        f_MessageSet(_stMsg);
      END_IF
    END_IF
END_CASE
//---------------------------------------------------------------------------------------
//  get config data
//    - NCI: X,Y,Z and helper axis Ids
//---------------------------------------------------------------------------------------
CASE _eState
OF
  E_PROGRESS.PROGRESS_BUSY:
    _AxisIdentity             := _stConfiguration.PortalConfig.AxisIdentity;
    _eState                   := E_PROGRESS.PROGRESS_PREPARE;
END_CASE
//---------------------------------------------------------------------------------------
//  check config data and initialize NCI Group
//    --> ST_AXIS_GROUP_INFO: data struct for plausibility checks on NCI Group
//---------------------------------------------------------------------------------------
CASE _eState
OF
  E_PROGRESS.PROGRESS_PREPARE:
    _eRslt                    := Unit_StartUp(TRUE);
    
    IF (_eRslt = E_PROGRESS.PROGRESS_ERROR)
    THEN
      // base class did the messaging
      // exit with error
      _eStateError            := _eState;
      _eState                 := E_PROGRESS.PROGRESS_ERROR;
      _eRslt                  := Unit_StartUp(FALSE);   // clear method

    ELSIF (_eRslt = E_PROGRESS.PROGRESS_DONE)
    THEN
      // startup of NCI successful
      // next states are intended for customization
      _eState                 := E_PROGRESS.PROGRESS_STARTUP;
      _eRslt                  := Unit_StartUp(FALSE);   // clear method
    END_IF
END_CASE
//---------------------------------------------------------------------------------------
//---------------------------------------------------------------------------------------
CASE _eState
OF
  E_PROGRESS.PROGRESS_STARTUP:
      // simply an inexpensive placeholder to customize initialization to your needs
      _eState                 := E_PROGRESS.PROGRESS_CHECK;
END_CASE
//---------------------------------------------------------------------------------------
//---------------------------------------------------------------------------------------
CASE _eState
OF
  E_PROGRESS.PROGRESS_CHECK:
      _eState                 := E_PROGRESS.PROGRESS_OCCUPIED;
END_CASE
//---------------------------------------------------------------------------------------
//---------------------------------------------------------------------------------------
CASE _eState
OF
  E_PROGRESS.PROGRESS_OCCUPIED:
      _eState                 := E_PROGRESS.PROGRESS_WORKING;
END_CASE
//---------------------------------------------------------------------------------------
//---------------------------------------------------------------------------------------
CASE _eState
OF
  E_PROGRESS.PROGRESS_WORKING:
    _eState                   := E_PROGRESS.PROGRESS_DONE;

    IF (_MessageLevel > E_MessageType.eMessageError)
    THEN
      _stMsg.eType            := E_MessageType.eMessageInfo;
      _stMsg.eSubdevice       := e_Subdevice.JobControl_Init;
      _stMsg.iErrorNumber     := _eState;
      _stMsg.sText            := concat(': ', TO_STRING(_eState));
    
      f_MessageSet(_stMsg);
    END_IF
END_CASE


Job_Init                      := _eState;
END_METHOD

METHOD Job_Reset  : E_PROGRESS
VAR_INPUT
  Execute         : BOOL;
END_VAR
VAR_INST
  _eRslt,
  _eStateError,
  _eState         : E_PROGRESS;
END_VAR
//---------------------------------------------------------------------------------------
//---------------------------------------------------------------------------------------
IF NOT Execute THEN _eState   := _eStateError     := E_PROGRESS.PROGRESS_INIT;  RETURN; END_IF
//---------------------------------------------------------------------------------------
IF NOT Check() THEN Job_Reset := _eState          := E_PROGRESS.PROGRESS_ERROR; RETURN; END_IF
//---------------------------------------------------------------------------------------
//---------------------------------------------------------------------------------------
CASE _eState 
of
  E_PROGRESS.PROGRESS_INIT:
    IF Execute
    THEN
      _eState                 := E_PROGRESS.PROGRESS_BUSY;
      _eRslt                  := Unit_Reset(FALSE);   // clear method

      IF (_MessageLevel > E_MessageType.eMessageError)
      THEN
        _stMsg.eType          := E_MessageType.eMessageInfo;
        _stMsg.eSubdevice     := e_Subdevice.JobControl_Reset;
        _stMsg.iErrorNumber   := _eState;
        _stMsg.sText          := concat(': ', TO_STRING(_eState));
      
        f_MessageSet(_stMsg);
      END_IF
    END_IF
END_CASE
//---------------------------------------------------------------------------------------
//  clear axis and NCI
//    - NCI: X,Y,Z and helper axis Ids
//---------------------------------------------------------------------------------------
CASE _eState
OF
  E_PROGRESS.PROGRESS_BUSY:
    _eRslt                    := Unit_Reset(TRUE);
    
    IF (_eRslt = E_PROGRESS.PROGRESS_ERROR)
    THEN
      // base class did the messaging
      // exit with error
      _eStateError            := _eState;
      _eState                 := E_PROGRESS.PROGRESS_ERROR;
      _eRslt                  := Unit_Reset(FALSE);   // clear method

    ELSIF (_eRslt = E_PROGRESS.PROGRESS_DONE)
    THEN
      // reset of axis and NCI successful
      // next states are intended for customization
      _eState                 := E_PROGRESS.PROGRESS_STARTUP;
      _eRslt                  := Unit_Reset(FALSE);   // clear method
    END_IF
END_CASE
//---------------------------------------------------------------------------------------
//---------------------------------------------------------------------------------------
CASE _eState
OF
  E_PROGRESS.PROGRESS_PREPARE:
      // simply an inexpensive placeholder to customize initialization to your needs
      _eState                 := E_PROGRESS.PROGRESS_STARTUP;
END_CASE
//---------------------------------------------------------------------------------------
//---------------------------------------------------------------------------------------
CASE _eState
OF
  E_PROGRESS.PROGRESS_STARTUP:
      // simply an inexpensive placeholder to customize initialization to your needs
      _eState                 := E_PROGRESS.PROGRESS_CHECK;
END_CASE
//---------------------------------------------------------------------------------------
//---------------------------------------------------------------------------------------
CASE _eState
OF
  E_PROGRESS.PROGRESS_CHECK:
      _eState                 := E_PROGRESS.PROGRESS_OCCUPIED;
END_CASE
//---------------------------------------------------------------------------------------
//---------------------------------------------------------------------------------------
CASE _eState
OF
  E_PROGRESS.PROGRESS_OCCUPIED:
      _eState                 := E_PROGRESS.PROGRESS_WORKING;
END_CASE
//---------------------------------------------------------------------------------------
//---------------------------------------------------------------------------------------
CASE _eState
OF
  E_PROGRESS.PROGRESS_WORKING:
    _eState                   := E_PROGRESS.PROGRESS_DONE;

    IF (_MessageLevel > E_MessageType.eMessageError)
    THEN
      _stMsg.eType            := E_MessageType.eMessageInfo;
      _stMsg.eSubdevice       := e_Subdevice.JobControl_Reset;
      _stMsg.iErrorNumber     := _eState;
      _stMsg.sText            := concat(': ', TO_STRING(_eState));
    
      f_MessageSet(_stMsg);
    END_IF
END_CASE


Job_Reset                     := _eState;
END_METHOD

METHOD Job_Rinse  : E_PROGRESS
VAR_INPUT
  Execute         : BOOL;
END_VAR
VAR_INST
  _eRslt,
  _eStateError,
  _eState         : E_PROGRESS;
END_VAR
//---------------------------------------------------------------------------------------
//---------------------------------------------------------------------------------------
IF NOT Execute THEN _eState   := _eStateError     := E_PROGRESS.PROGRESS_INIT;  RETURN; END_IF
//---------------------------------------------------------------------------------------
IF NOT Check() THEN Job_Rinse := _eState          := E_PROGRESS.PROGRESS_ERROR; RETURN; END_IF
//---------------------------------------------------------------------------------------
//---------------------------------------------------------------------------------------
CASE _eState 
of
  E_PROGRESS.PROGRESS_INIT:
    IF Execute
    THEN
      _eState                 := E_PROGRESS.PROGRESS_BUSY;
      // get job data at start
      _JobData                := _stConfiguration.JobConfig.ParameterRinse;
      _eRslt                  := Unit_Job(FALSE, _JobData);   // clear method

      IF (_MessageLevel > E_MessageType.eMessageError)
      THEN
        _stMsg.eType          := E_MessageType.eMessageInfo;
        _stMsg.eSubdevice     := e_Subdevice.JobControl_Rinse;
        _stMsg.iErrorNumber   := _eState;
        _stMsg.sText          := concat(': ', TO_STRING(_eState));
      
        f_MessageSet(_stMsg);
      END_IF
    END_IF
END_CASE
//---------------------------------------------------------------------------------------
//  move PtP axis
//    - X,Y,Z
//---------------------------------------------------------------------------------------
CASE _eState
OF
  E_PROGRESS.PROGRESS_BUSY:
    _eRslt                    := Unit_Job(TRUE, _JobData);
    
    IF (_eRslt = E_PROGRESS.PROGRESS_ERROR)
    THEN
      // base class did the messaging
      // exit with error
      _eStateError            := _eState;
      _eState                 := E_PROGRESS.PROGRESS_ERROR;
      _eRslt                  := Unit_Job(FALSE, _JobData);   // clear method

    ELSIF (_eRslt = E_PROGRESS.PROGRESS_DONE)
    THEN
      // move of axis to home positions successful
      // next states are intended for customization
      _eState                 := E_PROGRESS.PROGRESS_STARTUP;
      _eRslt                  := Unit_Job(FALSE, _JobData);   // clear method
    END_IF
END_CASE
//---------------------------------------------------------------------------------------
//---------------------------------------------------------------------------------------
CASE _eState
OF
  E_PROGRESS.PROGRESS_PREPARE:
      // simply an inexpensive placeholder to customize initialization to your needs
      _eState                 := E_PROGRESS.PROGRESS_STARTUP;
END_CASE
//---------------------------------------------------------------------------------------
//---------------------------------------------------------------------------------------
CASE _eState
OF
  E_PROGRESS.PROGRESS_STARTUP:
      // simply an inexpensive placeholder to customize initialization to your needs
      _eState                 := E_PROGRESS.PROGRESS_CHECK;
END_CASE
//---------------------------------------------------------------------------------------
//---------------------------------------------------------------------------------------
CASE _eState
OF
  E_PROGRESS.PROGRESS_CHECK:
      _eState                 := E_PROGRESS.PROGRESS_OCCUPIED;
END_CASE
//---------------------------------------------------------------------------------------
//---------------------------------------------------------------------------------------
CASE _eState
OF
  E_PROGRESS.PROGRESS_OCCUPIED:
      _eState                 := E_PROGRESS.PROGRESS_WORKING;
END_CASE
//---------------------------------------------------------------------------------------
//---------------------------------------------------------------------------------------
CASE _eState
OF
  E_PROGRESS.PROGRESS_WORKING:
    _eState                   := E_PROGRESS.PROGRESS_DONE;

    IF (_MessageLevel > E_MessageType.eMessageError)
    THEN
      _stMsg.eType            := E_MessageType.eMessageInfo;
      _stMsg.eSubdevice       := e_Subdevice.JobControl_Rinse;
      _stMsg.iErrorNumber     := _eState;
      _stMsg.sText            := concat(': ', TO_STRING(_eState));
    
      f_MessageSet(_stMsg);
    END_IF
END_CASE


Job_Rinse                     := _eState;
END_METHOD

PROPERTY State : reference to ST_JOB_STATE
SET
_stState ref= State;
END_SET
END_PROPERTY

END_FUNCTION_BLOCK

// ---- APPLICATION/JOB_CONTROL/fb_JobBase.TcPOU
//---------------------------------------------------------------------------------------------------------------
//
//  HAUD 2026.09.01
//  - PLC_MOTION_LAYER
//
//  fb_JobBase
//  - facilitates coordination of NCI 3D Group and PtP axis
//  - config 3D Group for NCI portal
//  - startup axis and NCI portal
//  - init and reset for error quit
//  - command ptp movement to Job starting positions (Home, Meas, Rinse, Weigh)
//  - command NCI config in Unit_Startup()
//
//
//---------------------------------------------------------------------------------------------------------------
// This SOFTWARE is provided as an Example by THE PROVIDER "as is" and "with all faults." THE PROVIDER makes no 
// representations or warranties of any kind concerning the safety, suitability, lack of viruses, inaccuracies, 
// typographical errors, or other harmful components of this SOFTWARE. There are inherent dangers in the use of 
// any software, and you are solely responsible for determining whether this SOFTWARE is compatible with your 
// equipment and other software installed on your equipment. You are also solely responsible for the protection 
// of your equipment and backup of your data, and THE PROVIDER will not be liable for any damages you may suffer 
// in connection with using, modifying, or distributing this SOFTWARE.
//---------------------------------------------------------------------------------------------------------------
FUNCTION_BLOCK ABSTRACT fb_JobBase
VAR
  _eCheck             : E_JOB_CHECK;

  _eResult            : E_PROGRESS;
  _eInit              : E_PROGRESS;

  _Blocked            : BOOL;   // flow control may use this for breaks during execution

  _rOverrideAxis      : LREAL := 100.0;
  _rOverrideChannel   : LREAL := 100.0;

  _AxisCtrl           : REFERENCE TO ARRAY[1..MAX_AXIS] OF ST_AXIS_CTRL;
  _AxisState          : REFERENCE TO ARRAY[1..MAX_AXIS] OF ST_AXIS_STATE;
  _AxisInfo           : REFERENCE TO ARRAY[1..MAX_AXIS] OF ST_AXIS_INFO;
  _AxisMoveData       : REFERENCE TO ARRAY[1..MAX_AXIS] OF ST_MOVE_DATA;

  _AxisIdentity       : REFERENCE TO ST_3D_Group;                         // NC Axis Id required for building 3D Group in NCI. You have to configure this
  _AxisGroupInfo      : ARRAY[1..NCI_AXIS_COUNT] OF ST_AXIS_GROUP_INFO;   // indices for batch processing of NC axis, entry carries index and NC Id

  _ChannelCtrl        : REFERENCE TO ST_NCI_CTRL;
  _ChannelState       : REFERENCE TO ST_NCI_STATE;

  _JobData            : ST_JOB_PARAMETER;   // job detail has to be written by extending class

  _eDeviceId          : e_Device;           // whoami?
  _MessageLevel       : E_MessageType;      // how much to tell?
  _stMsg              : ST_Message;
END_VAR
VAR CONSTANT
  X                   : UINT := 1;
  Y                   : UINT := 2;
  Z                   : UINT := 3;
  NCI_AXIS_COUNT      : UINT := 8;
END_VAR

PROPERTY AxisCtrl : reference TO ARRAY[1..MAX_AXIS] OF ST_AXIS_CTRL
SET
_AxisCtrl REF= AxisCtrl;
END_SET
END_PROPERTY

PROPERTY AxisInfo : reference TO ARRAY[1..MAX_AXIS] OF ST_AXIS_INFO
SET
_AxisInfo ref= AxisInfo;
END_SET
END_PROPERTY

PROPERTY AxisOverride : lreal
GET
AxisOverride := _rOverrideAxis;
END_GET
SET
_rOverrideAxis := AxisOverride;
END_SET
END_PROPERTY

PROPERTY AxisState : reference TO ARRAY[1..MAX_AXIS] OF ST_AXIS_STATE
SET
_AxisState ref= AxisState;
END_SET
END_PROPERTY

METHOD PROTECTED CheckBase : BOOL

IF NOT __isvalidref(_AxisCtrl)
THEN
  _eResult                          := E_PROGRESS.PROGRESS_ERROR;
  _eCheck                           := E_JOB_CHECK.POINTER_NULL_AXIS_CTRL;
  RETURN;
END_IF

IF NOT __ISVALIDREF(_AxisState)
THEN
  _eResult                          := E_PROGRESS.PROGRESS_ERROR;
  _eCheck                           := E_JOB_CHECK.POINTER_NULL_AXIS_STATE;
  RETURN;
END_IF

IF NOT __ISVALIDREF(_AxisInfo)
THEN
  _eResult                          := E_PROGRESS.PROGRESS_ERROR;
  _eCheck                           := E_JOB_CHECK.POINTER_NULL_AXIS_INFO;
  RETURN;
END_IF

IF NOT __ISVALIDREF(_AxisMoveData)
THEN
  _eResult                          := E_PROGRESS.PROGRESS_ERROR;
  _eCheck                           := E_JOB_CHECK.POINTER_NULL_AXIS_MOVE_DATA;
  RETURN;
END_IF

IF NOT __ISVALIDREF(_AxisIdentity)
THEN
  _eResult                          := E_PROGRESS.PROGRESS_ERROR;
  _eCheck                           := E_JOB_CHECK.POINTER_NULL_AXIS_IDENTITY;
  RETURN;
END_IF

IF NOT __ISVALIDREF(_ChannelCtrl)
THEN
  _eResult                          := E_PROGRESS.PROGRESS_ERROR;
  _eCheck                           := E_JOB_CHECK.POINTER_NULL_NCI_CHN_CTRL;
  RETURN;
END_IF

IF NOT __ISVALIDREF(_ChannelState)
THEN
  _eResult                          := E_PROGRESS.PROGRESS_ERROR;
  _eCheck                           := E_JOB_CHECK.POINTER_NULL_NCI_CHN_STATE;
  RETURN;
END_IF

_eCheck                             := E_JOB_CHECK.CHECK_DONE;
CheckBase                           := TRUE;
END_METHOD

PROPERTY ChnAxisIdentity : reference TO ST_3D_Group
SET
_AxisIdentity ref= ChnAxisIdentity;
END_SET
END_PROPERTY

PROPERTY ChnCtrl : reference TO ST_NCI_CTRL
SET
_ChannelCtrl ref= ChnCtrl;
END_SET
END_PROPERTY

PROPERTY ChnOverride : lreal
GET
ChnOverride := _rOverrideChannel;
END_GET
SET
_rOverrideChannel := ChnOverride;
END_SET
END_PROPERTY

PROPERTY ChnState : reference TO ST_NCI_STATE
SET
_ChannelState ref= ChnState;
END_SET
END_PROPERTY

METHOD PRIVATE GetGroupIndices : e_progress // TC2 NCI - get indices for 8 Axis[] from ChnAxisIdentity(ST_3D_GROUP); X,Y,Z,Q1,Q2,Q3,Q4,Q5
VAR_INPUT
  Execute     : BOOL;
END_VAR
VAR_INST
  _idx, _idy  : UDINT;
  _nState     : E_PROGRESS;
  _nAxisId    : ARRAY[1..NCI_AXIS_COUNT] OF ST_AXIS_GROUP_INFO; // 8 is the magic number, just as in the TC2 NCI
  _wValid     : DWORD;
END_VAR
IF NOT Execute THEN _nState         := E_PROGRESS.PROGRESS_INIT; END_IF
IF NOT CheckBase() THEN GetGroupIndices := E_PROGRESS.PROGRESS_ERROR; END_IF
//---------------------------------------------------------------------------------------------------------------
CASE _nState 
OF
  //-------------------------------------------------------------------------------------------------------------
  E_PROGRESS.PROGRESS_INIT:
    IF Execute
    THEN
      _nState                           := E_PROGRESS.PROGRESS_BUSY;

      memset(ADR(_wValid),        0, SIZEOF(_wValid));
      memset(ADR(_nAxisId),       0, SIZEOF(_nAxisId));
      memset(ADR(_AxisGroupInfo), 0, SIZEOF(_AxisGroupInfo));

      _nAxisId[1].bHasValue             := (_AxisIdentity.nXAxisId  > 0);
      _nAxisId[1].nAxisId               :=  _AxisIdentity.nXAxisId;
      _nAxisId[1].bMainAxis             := TRUE;

      _nAxisId[2].bHasValue             := (_AxisIdentity.nYAxisId  > 0);
      _nAxisId[2].nAxisId               :=  _AxisIdentity.nYAxisId;
      _nAxisId[2].bMainAxis             := TRUE;

      _nAxisId[3].bHasValue             := (_AxisIdentity.nZAxisId  > 0);
      _nAxisId[3].nAxisId               :=  _AxisIdentity.nZAxisId;
      _nAxisId[3].bMainAxis             := TRUE;

      _nAxisId[4].bHasValue             := (_AxisIdentity.nQ1AxisId > 0);
      _nAxisId[4].nAxisId               :=  _AxisIdentity.nQ1AxisId;

      _nAxisId[5].bHasValue             := (_AxisIdentity.nQ2AxisId > 0);
      _nAxisId[5].nAxisId               :=  _AxisIdentity.nQ2AxisId;

      _nAxisId[6].bHasValue             := (_AxisIdentity.nQ3AxisId > 0);
      _nAxisId[6].nAxisId               :=  _AxisIdentity.nQ3AxisId;

      _nAxisId[7].bHasValue             := (_AxisIdentity.nQ4AxisId > 0);
      _nAxisId[7].nAxisId               :=  _AxisIdentity.nQ4AxisId;

      _nAxisId[8].bHasValue             := (_AxisIdentity.nQ5AxisId > 0);
      _nAxisId[8].nAxisId               :=  _AxisIdentity.nQ5AxisId;
    END_IF
END_CASE
//---------------------------------------------------------------------------------------------------------------
CASE _nState 
OF
  //-------------------------------------------------------------------------------------------------------------
  E_PROGRESS.PROGRESS_BUSY:
    _nState                             := E_PROGRESS.PROGRESS_PREPARE;
    FOR _idx := 1 TO NCI_AXIS_COUNT
    DO
      IF (_nAxisId[_idx].bHasValue)
      THEN
        FOR _idy := 1 TO PLC_CONSTANT.MAX_AXIS
        DO
          IF (_nAxisId[_idx].nAxisId = _AxisInfo[_idy].nNcAxisId)
          THEN
            _nAxisId[_idx].nAxisIndex   := _idy;
            _nAxisId[_idx].bValid       := TRUE;
            EXIT;
          END_IF
        END_FOR
      END_IF
    END_FOR
END_CASE
//---------------------------------------------------------------------------------------------------------------
CASE _nState 
OF
  //-------------------------------------------------------------------------------------------------------------
  E_PROGRESS.PROGRESS_PREPARE:
    _nState                             := E_PROGRESS.PROGRESS_WORKING;
    FOR _idx := 1 TO 8
    DO
      IF (_nAxisId[_idx].bValid)
      THEN
        _wValid                         := Tc2_System.SETBIT32(_wValid, TO_SINT(_idx-1));
      END_IF
    END_FOR
END_CASE
//---------------------------------------------------------------------------------------------------------------
CASE _nState 
OF
  //-------------------------------------------------------------------------------------------------------------
  E_PROGRESS.PROGRESS_WORKING:
    IF (_wValid > 0)
    THEN
      _nState                           := E_PROGRESS.PROGRESS_DONE;
    ELSE
      _nState                           := E_PROGRESS.PROGRESS_ERROR;
    END_IF

    _AxisGroupInfo                      := _nAxisId;
END_CASE
//---------------------------------------------------------------------------------------------------------------
GetGroupIndices                         := _nState;
//---------------------------------------------------------------------------------------------------------------
END_METHOD

METHOD Unit_Job : e_progress
VAR_INPUT
  Execute       : BOOL;
  JobParameter  : ST_JOB_PARAMETER;
END_VAR
VAR_INST
  _nSubState,
  _nResult,
  _nState       : e_progress;

  _nErrorId     : UDINT;
  _idx          : UINT;
END_VAR
//---------------------------------------------------------------------------------------------------------------
//---------------------------------------------------------------------------------------------------------------
IF NOT Execute THEN _nState           := E_PROGRESS.PROGRESS_INIT; END_IF
//---------------------------------------------------------------------------------------------------------------
IF NOT CheckBase() THEN Unit_Job      := E_PROGRESS.PROGRESS_ERROR; RETURN; END_IF
//---------------------------------------------------------------------------------------------------------------
//---------------------------------------------------------------------------------------------------------------
CASE _nState 
OF
  E_PROGRESS.PROGRESS_INIT:
    IF Execute
    THEN
      _idx                            := 1;
      _nSubState                      := E_PROGRESS.PROGRESS_INIT;
      _nState                         := E_PROGRESS.PROGRESS_BUSY;

      IF (_MessageLevel > E_MessageType.eMessageError)
      THEN
        _stMsg.eType                  := E_MessageType.eMessageInfo;
        _stMsg.eSubdevice             := e_Subdevice.JobBase_Job;
        _stMsg.iErrorNumber           := 0;
        _stMsg.sText                  := concat(' : ', TO_STRING(_nState));

        f_MessageSet(_stMsg);
      END_IF
    END_IF
END_CASE
//---------------------------------------------------------------------------------------------------------------
CASE _nState 
OF
  E_PROGRESS.PROGRESS_BUSY:
    CASE _nSubState
    OF
      //---------------------------------------------------------------------------
      E_PROGRESS.PROGRESS_INIT:
        IF NOT (_AxisGroupInfo[_idx].bValid)
        THEN
          _nSubState                  := E_PROGRESS.PROGRESS_BUSY;
        ELSE
          _AxisCtrl[_AxisGroupInfo[_idx].nAxisIndex].eCmd        := E_AXIS_CTRL.AXIS_ENABLE;
    
          IF (_AxisState[_AxisGroupInfo[_idx].nAxisIndex].eState = E_AXIS_STATE.AXIS_ENABLE + E_PROGRESS.PROGRESS_DONE)
          THEN
            _nSubState                := E_PROGRESS.PROGRESS_BUSY;

            IF (_MessageLevel > E_MessageType.eMessageWarning)
            THEN
              _stMsg.eType            := E_MessageType.eMessageInfo;
              _stMsg.eSubdevice       := e_Subdevice.JobBase_Job;
              _stMsg.iErrorNumber     := _AxisGroupInfo[_idx].nAxisId;
              _stMsg.sText            := concat('AXIS_ENABLE: ', TO_STRING(E_PROGRESS.PROGRESS_DONE));
        
              f_MessageSet(_stMsg);
            END_IF
          END_IF
        END_IF

      //---------------------------------------------------------------------------
      E_PROGRESS.PROGRESS_BUSY:
        IF (_idx > NCI_AXIS_COUNT-1)
        THEN
          _idx                        := 1;
          _nSubState                  := E_PROGRESS.PROGRESS_INIT;
          _nState                     := E_PROGRESS.PROGRESS_PREPARE;
        ELSE
          _idx                        := _idx + 1;
          _nSubState                  := E_PROGRESS.PROGRESS_INIT;
        END_IF
    END_CASE
END_CASE
//---------------------------------------------------------------------------------------------------------------
CASE _nState 
OF
  //---------------------------------------------------------------------------
  E_PROGRESS.PROGRESS_PREPARE:
    CASE _nSubState
    OF
      //-----------------------------------------------------------------------
      E_PROGRESS.PROGRESS_INIT:
        IF NOT (_AxisGroupInfo[_idx].bValid)
        THEN
          _nSubState                  := E_PROGRESS.PROGRESS_BUSY;
        ELSE
          _AxisCtrl[_AxisGroupInfo[_idx].nAxisIndex].eCmd        := E_AXIS_CTRL.AXIS_RESET;
    
          IF (_AxisState[_AxisGroupInfo[_idx].nAxisIndex].eState = E_AXIS_STATE.AXIS_RESET + E_PROGRESS.PROGRESS_DONE)
          THEN
            _nSubState                := E_PROGRESS.PROGRESS_BUSY;

            IF (_MessageLevel > E_MessageType.eMessageWarning)
            THEN
              _stMsg.eType            := E_MessageType.eMessageInfo;
              _stMsg.eSubdevice       := e_Subdevice.JobBase_Job;
              _stMsg.iErrorNumber     := _AxisGroupInfo[_idx].nAxisId;
              _stMsg.sText            := concat('AXIS_RESET: ', TO_STRING(E_PROGRESS.PROGRESS_DONE));
        
              f_MessageSet(_stMsg);
            END_IF
          END_IF
        END_IF
      //-----------------------------------------------------------------------
      E_PROGRESS.PROGRESS_BUSY:
        IF (_idx > NCI_AXIS_COUNT-1)
        THEN
          _idx                        := 1;
          _nSubState                  := E_PROGRESS.PROGRESS_INIT;
          _nState                     := E_PROGRESS.PROGRESS_STARTUP;
        ELSE
          _idx                        := _idx + 1;
          _nSubState                  := E_PROGRESS.PROGRESS_INIT;
        END_IF
    END_CASE

  //---------------------------------------------------------------------------
  E_PROGRESS.PROGRESS_STARTUP:
    CASE _nSubState
    OF
      //-----------------------------------------------------------------------
      E_PROGRESS.PROGRESS_INIT:
        _ChannelCtrl.eCmd            := E_NCI_CTRL.INIT;
        _nSubState                    := E_PROGRESS.PROGRESS_BUSY;
      //-----------------------------------------------------------------------
      E_PROGRESS.PROGRESS_BUSY:
        IF (_ChannelState.eState = E_NCI_STATE.INIT + E_PROGRESS.PROGRESS_DONE)
        THEN
          _idx                        := 1;
          _nSubState                  := E_PROGRESS.PROGRESS_INIT;
          _nState                     := E_PROGRESS.PROGRESS_CHECK;

          IF (_MessageLevel > E_MessageType.eMessageWarning)
          THEN
            _stMsg.eType              := E_MessageType.eMessageInfo;
            _stMsg.eSubdevice         := e_Subdevice.JobBase_Job;
            _stMsg.iErrorNumber       := _ChannelState.eState;
            _stMsg.sText              := concat('E_NCI_CTRL.INIT: ', TO_STRING(E_PROGRESS.PROGRESS_DONE));
      
            f_MessageSet(_stMsg);
          END_IF
        END_IF
    END_CASE
  //---------------------------------------------------------------------------
  E_PROGRESS.PROGRESS_CHECK:
    CASE _nSubState
    OF
      //-----------------------------------------------------------------------
      E_PROGRESS.PROGRESS_INIT:
        _nSubState                    := E_PROGRESS.PROGRESS_BUSY;

        _AxisMoveData[_AxisGroupInfo[Z].nAxisIndex].rSetPos    := JobParameter.CollisionZ;   // move up z-axis to collision free position, in order to move X,Y axis safely.
        _AxisMoveData[_AxisGroupInfo[Z].nAxisIndex].rSetVelo   := JobParameter.DynConstraint[Z].rSetVelo;
        _AxisMoveData[_AxisGroupInfo[Z].nAxisIndex].rAcc       := JobParameter.DynConstraint[Z].rAcc;
        _AxisMoveData[_AxisGroupInfo[Z].nAxisIndex].rDec       := JobParameter.DynConstraint[Z].rDec;
        _AxisMoveData[_AxisGroupInfo[Z].nAxisIndex].rOverride  := _rOverrideAxis;

      //-----------------------------------------------------------------------
      E_PROGRESS.PROGRESS_BUSY:
        _AxisCtrl    [_AxisGroupInfo[Z].nAxisIndex].eCmd       := E_AXIS_CTRL.AXIS_MOVE_POS;

        IF (_AxisState[_AxisGroupInfo[Z].nAxisIndex].eState = E_AXIS_STATE.AXIS_MOVE_POS + E_PROGRESS.PROGRESS_ERROR)
        THEN
          _nState                     := E_PROGRESS.PROGRESS_ERROR;

          _stMsg.eType                := E_MessageType.eMessageError;
          _stMsg.eSubdevice           := e_Subdevice.JobBase_Job;
          _stMsg.iErrorNumber         := _AxisGroupInfo[Z].nAxisId;
          _stMsg.sText                := concat('Z-AXIS_MOVE_POS: ', TO_STRING(_nState));
          f_MessageSet(_stMsg);

        ELSIF (_AxisState[_AxisGroupInfo[Z].nAxisIndex].eState = E_AXIS_STATE.AXIS_MOVE_POS + E_PROGRESS.PROGRESS_DONE)
        THEN
          _nSubState                  := E_PROGRESS.PROGRESS_PREPARE;
        END_IF

      //-----------------------------------------------------------------------
      E_PROGRESS.PROGRESS_PREPARE:
        _nSubState                    := E_PROGRESS.PROGRESS_STARTUP;

        _AxisMoveData[_AxisGroupInfo[X].nAxisIndex].rSetPos    := JobParameter.Position.x;
        _AxisMoveData[_AxisGroupInfo[X].nAxisIndex].rSetVelo   := JobParameter.DynConstraint[X].rSetVelo;
        _AxisMoveData[_AxisGroupInfo[X].nAxisIndex].rAcc       := JobParameter.DynConstraint[X].rAcc;
        _AxisMoveData[_AxisGroupInfo[X].nAxisIndex].rDec       := JobParameter.DynConstraint[X].rDec;
        _AxisMoveData[_AxisGroupInfo[X].nAxisIndex].rOverride  := _rOverrideAxis;

        _AxisMoveData[_AxisGroupInfo[Y].nAxisIndex].rSetPos    := JobParameter.Position.Y;
        _AxisMoveData[_AxisGroupInfo[Y].nAxisIndex].rSetVelo   := JobParameter.DynConstraint[Y].rSetVelo;
        _AxisMoveData[_AxisGroupInfo[Y].nAxisIndex].rAcc       := JobParameter.DynConstraint[Y].rAcc;
        _AxisMoveData[_AxisGroupInfo[Y].nAxisIndex].rDec       := JobParameter.DynConstraint[Y].rDec;
        _AxisMoveData[_AxisGroupInfo[Y].nAxisIndex].rOverride  := _rOverrideAxis;

      //-----------------------------------------------------------------------
      E_PROGRESS.PROGRESS_STARTUP:
        _AxisCtrl    [_AxisGroupInfo[X].nAxisIndex].eCmd       := E_AXIS_CTRL.AXIS_MOVE_POS;
        _AxisCtrl    [_AxisGroupInfo[Y].nAxisIndex].eCmd       := E_AXIS_CTRL.AXIS_MOVE_POS;

        IF (_AxisState[_AxisGroupInfo[X].nAxisIndex].eState = E_AXIS_STATE.AXIS_MOVE_POS + E_PROGRESS.PROGRESS_ERROR) OR
           (_AxisState[_AxisGroupInfo[Y].nAxisIndex].eState = E_AXIS_STATE.AXIS_MOVE_POS + E_PROGRESS.PROGRESS_ERROR)
        THEN
          _nState                     := E_PROGRESS.PROGRESS_ERROR;

          _stMsg.eType                := E_MessageType.eMessageError;
          _stMsg.eSubdevice           := e_Subdevice.NciJob;

          IF (_AxisState[_AxisGroupInfo[X].nAxisIndex].eState = E_AXIS_STATE.AXIS_MOVE_POS + E_PROGRESS.PROGRESS_ERROR)
          THEN
            _stMsg.iErrorNumber       := _AxisGroupInfo[X].nAxisId;
            _stMsg.sText              := concat('X-AXIS_MOVE_POS: ', TO_STRING(_nState));
          ELSE
            _stMsg.iErrorNumber       := _AxisGroupInfo[Y].nAxisId;
            _stMsg.sText              := concat('Y-AXIS_MOVE_POS: ', TO_STRING(_nState));
          END_IF

          f_MessageSet(_stMsg);

        ELSE
          IF (_AxisState[_AxisGroupInfo[X].nAxisIndex].eState = E_AXIS_STATE.AXIS_MOVE_POS + E_PROGRESS.PROGRESS_DONE) AND
             (_AxisState[_AxisGroupInfo[Y].nAxisIndex].eState = E_AXIS_STATE.AXIS_MOVE_POS + E_PROGRESS.PROGRESS_DONE)
          THEN
            _nSubState                := E_PROGRESS.PROGRESS_CHECK;
          END_IF
        END_IF

      //-----------------------------------------------------------------------
      E_PROGRESS.PROGRESS_CHECK:
        _nSubState                    := E_PROGRESS.PROGRESS_OCCUPIED;

        _AxisMoveData[_AxisGroupInfo[Z].nAxisIndex].rSetPos    := JobParameter.Position.z;   // move z-axis to final position
        _AxisMoveData[_AxisGroupInfo[Z].nAxisIndex].rSetVelo   := JobParameter.DynConstraint[Z].rSetVelo;
        _AxisMoveData[_AxisGroupInfo[Z].nAxisIndex].rAcc       := JobParameter.DynConstraint[Z].rAcc;
        _AxisMoveData[_AxisGroupInfo[Z].nAxisIndex].rDec       := JobParameter.DynConstraint[Z].rDec;
        _AxisMoveData[_AxisGroupInfo[Z].nAxisIndex].rOverride  := _rOverrideAxis;

      //-----------------------------------------------------------------------
      E_PROGRESS.PROGRESS_OCCUPIED:
        _AxisCtrl    [_AxisGroupInfo[Z].nAxisIndex].eCmd       := E_AXIS_CTRL.AXIS_MOVE_POS;

        IF (_AxisState[_AxisGroupInfo[Z].nAxisIndex].eState = E_AXIS_STATE.AXIS_MOVE_POS + E_PROGRESS.PROGRESS_ERROR)
        THEN
          _nState                     := E_PROGRESS.PROGRESS_ERROR;

          _stMsg.eType                := E_MessageType.eMessageError;
          _stMsg.eSubdevice           := e_Subdevice.JobBase_Job;
          _stMsg.iErrorNumber         := _AxisGroupInfo[Z].nAxisId;
          _stMsg.sText                := concat('Z-AXIS_MOVE_POS: ', TO_STRING(_nState));
          f_MessageSet(_stMsg);

        ELSIF (_AxisState[_AxisGroupInfo[Z].nAxisIndex].eState = E_AXIS_STATE.AXIS_MOVE_POS + E_PROGRESS.PROGRESS_DONE)
        THEN
          _nSubState                  := E_PROGRESS.PROGRESS_INIT;
          _nState                     := E_PROGRESS.PROGRESS_OCCUPIED;
        END_IF
    END_CASE
END_CASE
//---------------------------------------------------------------------------------------------------------------
CASE _nState 
OF
  //---------------------------------------------------------------------------
  E_PROGRESS.PROGRESS_OCCUPIED:
    _nState                           := E_PROGRESS.PROGRESS_DONE;
END_CASE
//---------------------------------------------------------------------------------------------------------------
Unit_Job                              := _nState;
//---------------------------------------------------------------------------------------------------------------
END_METHOD

METHOD Unit_Reset : e_progress
VAR_INPUT
  Execute       : BOOL;
END_VAR
VAR_INST
  _nSubState,
  _nResult,
  _nState       : e_progress;

  _nErrorId     : UDINT;
  _idx          : UINT;
END_VAR
//---------------------------------------------------------------------------------------------------------------
//---------------------------------------------------------------------------------------------------------------
IF NOT Execute THEN _nState           := E_PROGRESS.PROGRESS_INIT; END_IF
//---------------------------------------------------------------------------------------------------------------
IF NOT CheckBase() THEN Unit_Reset    := E_PROGRESS.PROGRESS_ERROR; RETURN; END_IF
//---------------------------------------------------------------------------------------------------------------
//---------------------------------------------------------------------------------------------------------------
CASE _nState 
OF
  E_PROGRESS.PROGRESS_INIT:
    IF Execute
    THEN
      _idx                            := 1;
      _nSubState                      := E_PROGRESS.PROGRESS_INIT;
      _nState                         := E_PROGRESS.PROGRESS_BUSY;

      IF (_MessageLevel > E_MessageType.eMessageError)
      THEN
        _stMsg.eType                  := E_MessageType.eMessageInfo;
        _stMsg.eSubdevice             := e_Subdevice.JobBase_Reset;
        _stMsg.iErrorNumber           := 0;
        _stMsg.sText                  := concat(' : ', TO_STRING(_nState));

        f_MessageSet(_stMsg);
      END_IF

    END_IF
END_CASE
//-----------------------------------------------------------------------------
CASE _nState 
OF
  E_PROGRESS.PROGRESS_BUSY:
    CASE _nSubState
    OF
      E_PROGRESS.PROGRESS_INIT:
        IF NOT (_AxisGroupInfo[_idx].bValid)
        THEN
          _nSubState                  := E_PROGRESS.PROGRESS_BUSY;
        ELSE
          _AxisCtrl[_AxisGroupInfo[_idx].nAxisIndex].eCmd        := E_AXIS_CTRL.AXIS_RESET;
    
          IF (_AxisState[_AxisGroupInfo[_idx].nAxisIndex].eState = E_AXIS_STATE.AXIS_RESET + E_PROGRESS.PROGRESS_DONE)
          THEN
            _nSubState                := E_PROGRESS.PROGRESS_BUSY;

            IF (_MessageLevel > E_MessageType.eMessageWarning)
            THEN
              _stMsg.eType            := E_MessageType.eMessageInfo;
              _stMsg.eSubdevice       := e_Subdevice.JobBase_Reset;
              _stMsg.iErrorNumber     := _AxisGroupInfo[_idx].nAxisId;
              _stMsg.sText            := concat('AXIS_RESET: ', TO_STRING(E_PROGRESS.PROGRESS_DONE));
        
              f_MessageSet(_stMsg);
            END_IF
          END_IF
        END_IF

      E_PROGRESS.PROGRESS_BUSY:
        IF (_idx > NCI_AXIS_COUNT-1)
        THEN
          _idx                        := 1;
          _nSubState                  := E_PROGRESS.PROGRESS_INIT;
          _nState                     := E_PROGRESS.PROGRESS_STARTUP;
        ELSE
          _idx                        := _idx + 1;
          _nSubState                  := E_PROGRESS.PROGRESS_INIT;
        END_IF
    END_CASE
END_CASE
//-----------------------------------------------------------------------------
CASE _nState 
OF
  //---------------------------------------------------------------------------
  E_PROGRESS.PROGRESS_STARTUP:
    CASE _nSubState
    OF
      E_PROGRESS.PROGRESS_INIT:
        _ChannelCtrl.eCmd            := E_NCI_CTRL.RESET;
        _nSubState                    := E_PROGRESS.PROGRESS_BUSY;

      E_PROGRESS.PROGRESS_BUSY:
        IF (_ChannelState.eState = E_NCI_STATE.RESET + E_PROGRESS.PROGRESS_DONE)
        THEN
          _idx                        := 1;
          _nSubState                  := E_PROGRESS.PROGRESS_INIT;
          _nState                     := E_PROGRESS.PROGRESS_OCCUPIED;

          IF (_MessageLevel > E_MessageType.eMessageWarning)
          THEN
            _stMsg.eType              := E_MessageType.eMessageInfo;
            _stMsg.eSubdevice         := e_Subdevice.JobBase_Reset;
            _stMsg.iErrorNumber       := _ChannelState.eState;
            _stMsg.sText              := concat('E_NCI_CTRL.RESET: ', TO_STRING(E_PROGRESS.PROGRESS_DONE));
      
            f_MessageSet(_stMsg);
          END_IF
        END_IF
    END_CASE
END_CASE
//-----------------------------------------------------------------------------
CASE _nState 
OF
  //---------------------------------------------------------------------------
  E_PROGRESS.PROGRESS_OCCUPIED:
    _nState                           := E_PROGRESS.PROGRESS_DONE;
END_CASE
//-----------------------------------------------------------------------------
Unit_Reset                            := _nState;
//-----------------------------------------------------------------------------
END_METHOD

METHOD Unit_Startup : e_progress
VAR_INPUT
  Execute           : BOOL;
END_VAR
VAR_INST
  _nSubState,
  _nResult,
  _nState           : e_progress;

  _nErrorId         : UDINT;
  _idx              : UINT;
END_VAR
//---------------------------------------------------------------------------------------------------------------
//---------------------------------------------------------------------------------------------------------------
IF NOT Execute THEN _nState           := E_PROGRESS.PROGRESS_INIT; END_IF
//---------------------------------------------------------------------------------------------------------------
IF NOT CheckBase() THEN Unit_Startup  := E_PROGRESS.PROGRESS_ERROR; RETURN; END_IF
//---------------------------------------------------------------------------------------------------------------
//---------------------------------------------------------------------------------------------------------------
CASE _nState 
OF
  //-------------------------------------------------------------------------------------------------------------
  E_PROGRESS.PROGRESS_INIT:
    IF Execute
    THEN
      _idx                            := 1;
      _nResult                        := GetGroupIndices(FALSE);
      _nState                         := E_PROGRESS.PROGRESS_BUSY;

      IF (_MessageLevel > E_MessageType.eMessageError)
      THEN
        _stMsg.eType                  := E_MessageType.eMessageInfo;
        _stMsg.eSubdevice             := e_Subdevice.JobBase_StartUp;
        _stMsg.iErrorNumber           := 0;
        _stMsg.sText                  := concat(' : ', TO_STRING(_nState));
  
        f_MessageSet(_stMsg);
      END_IF
    END_IF
END_CASE
//---------------------------------------------------------------------------------------------------------------
CASE _nState
OF
  //-------------------------------------------------------------------------------------------------------------
  E_PROGRESS.PROGRESS_BUSY:
    // check NCI configuration
    _nResult                          := GetGroupIndices(TRUE);

    IF (_nResult = E_PROGRESS.PROGRESS_ERROR)
    THEN
      _nState                         := E_PROGRESS.PROGRESS_ERROR;

      _stMsg.eType                    := E_MessageType.eMessageError;
      _stMsg.eSubdevice               := e_Subdevice.JobBase_StartUp;
      _stMsg.iErrorNumber             := 0;
      _stMsg.sText                    := concat('GetGroupIndices: ', TO_STRING(_nResult));
      f_MessageSet(_stMsg);

      _nResult                        := GetGroupIndices(FALSE);

    ELSIF (_nResult = E_PROGRESS.PROGRESS_DONE)
    THEN
      _nSubState                      := E_PROGRESS.PROGRESS_INIT;
      _nState                         := E_PROGRESS.PROGRESS_PREPARE;

      IF (_MessageLevel > E_MessageType.eMessageWarning)
      THEN
        _stMsg.eType                  := E_MessageType.eMessageInfo;
        _stMsg.eSubdevice             := e_Subdevice.JobBase_StartUp;
        _stMsg.iErrorNumber           := 0;
        _stMsg.sText                  := concat('GetGroupIndices: ', TO_STRING(_nResult));
  
        f_MessageSet(_stMsg);
      END_IF

      _nResult                        := GetGroupIndices(FALSE);
    END_IF
END_CASE
//---------------------------------------------------------------------------------------------------------------
CASE _nState
OF
  //-------------------------------------------------------------------------------------------------------------
  E_PROGRESS.PROGRESS_PREPARE:
    CASE _nSubState
    OF
      E_PROGRESS.PROGRESS_INIT:
        IF NOT (_AxisGroupInfo[_idx].bValid)
        THEN
          _nSubState                  := E_PROGRESS.PROGRESS_BUSY;
        ELSE
          _AxisCtrl[_AxisGroupInfo[_idx].nAxisIndex].eCmd        := E_AXIS_CTRL.AXIS_DISABLE;
    
          IF (_AxisState[_AxisGroupInfo[_idx].nAxisIndex].eState = E_AXIS_STATE.AXIS_DISABLE + E_PROGRESS.PROGRESS_DONE)
          THEN
            _nSubState                := E_PROGRESS.PROGRESS_BUSY;

            IF (_MessageLevel > E_MessageType.eMessageWarning)
            THEN
              _stMsg.eType            := E_MessageType.eMessageInfo;
              _stMsg.eSubdevice       := e_Subdevice.JobBase_StartUp;
              _stMsg.iErrorNumber     := _AxisGroupInfo[_idx].nAxisId;
              _stMsg.sText            := concat('AXIS_DISABLE: ', TO_STRING(E_PROGRESS.PROGRESS_DONE));
        
              f_MessageSet(_stMsg);
            END_IF
          END_IF
        END_IF

      E_PROGRESS.PROGRESS_BUSY:
        IF (_idx > NCI_AXIS_COUNT-1)
        THEN
          _idx                        := 1;
          _nSubState                  := E_PROGRESS.PROGRESS_INIT;
          _nState                     := E_PROGRESS.PROGRESS_STARTUP;
        ELSE
          _idx                        := _idx + 1;
          _nSubState                  := E_PROGRESS.PROGRESS_INIT;
        END_IF
    END_CASE
  //-------------------------------------------------------------------------------------------------------------
  E_PROGRESS.PROGRESS_STARTUP:
    CASE _nSubState
    OF
      E_PROGRESS.PROGRESS_INIT:
        IF NOT (_AxisGroupInfo[_idx].bValid)
        THEN
          _nSubState                  := E_PROGRESS.PROGRESS_BUSY;
        ELSE
          _AxisCtrl[_AxisGroupInfo[_idx].nAxisIndex].eCmd       := E_AXIS_CTRL.AXIS_RESET;
      
          IF (_AxisState[_AxisGroupInfo[_idx].nAxisIndex].eState = E_AXIS_STATE.AXIS_RESET + E_PROGRESS.PROGRESS_ERROR)
          THEN
            _nState                   := E_PROGRESS.PROGRESS_ERROR;
      
              _stMsg.eType            := E_MessageType.eMessageError;
              _stMsg.eSubdevice       := e_Subdevice.JobBase_StartUp;
              _stMsg.iErrorNumber     := _AxisGroupInfo[_idx].nAxisId;
              _stMsg.sText            := concat('AXIS_RESET: ', TO_STRING(E_PROGRESS.PROGRESS_DONE));
        
              f_MessageSet(_stMsg);
      
          ELSIF (_AxisState[_AxisGroupInfo[_idx].nAxisIndex].eState = E_AXIS_STATE.AXIS_RESET + E_PROGRESS.PROGRESS_DONE)
          THEN
            _nState                   := E_PROGRESS.PROGRESS_BUSY;

            IF (_MessageLevel > E_MessageType.eMessageWarning)
            THEN
              _stMsg.eType            := E_MessageType.eMessageInfo;
              _stMsg.eSubdevice       := e_Subdevice.JobBase_StartUp;
              _stMsg.iErrorNumber     := _AxisGroupInfo[_idx].nAxisId;
              _stMsg.sText            := concat('AXIS_RESET: ', TO_STRING(E_PROGRESS.PROGRESS_DONE));
        
              f_MessageSet(_stMsg);
            END_IF
          END_IF
        END_IF

      E_PROGRESS.PROGRESS_BUSY:
        IF (_idx > NCI_AXIS_COUNT-1)
        THEN
          _idx                        := 1;
          _nSubState                  := E_PROGRESS.PROGRESS_INIT;
          _nState                     := E_PROGRESS.PROGRESS_CHECK;
        ELSE
          _idx                        := _idx + 1;
          _nSubState                  := E_PROGRESS.PROGRESS_INIT;
        END_IF
    END_CASE
  //-------------------------------------------------------------------------------------------------------------
  E_PROGRESS.PROGRESS_CHECK:
    CASE _nSubState
    OF
      E_PROGRESS.PROGRESS_INIT:
        _ChannelCtrl.eCmd             := E_NCI_CTRL.INIT;
        _nSubState                    := E_PROGRESS.PROGRESS_BUSY;

      E_PROGRESS.PROGRESS_BUSY:
        IF (_ChannelState.eState = E_NCI_STATE.INIT + E_PROGRESS.PROGRESS_DONE)
        THEN
          _nSubState                  := E_PROGRESS.PROGRESS_INIT;
          _nState                     := E_PROGRESS.PROGRESS_OCCUPIED;

          IF (_MessageLevel > E_MessageType.eMessageWarning)
          THEN
            _stMsg.eType              := E_MessageType.eMessageInfo;
            _stMsg.eSubdevice         := e_Subdevice.JobBase_StartUp;
            _stMsg.iErrorNumber       := _ChannelState.eState;
            _stMsg.sText              := concat('E_NCI_CTRL.INIT: ', TO_STRING(E_PROGRESS.PROGRESS_DONE));
      
            f_MessageSet(_stMsg);
          END_IF
        END_IF
    END_CASE
  //-------------------------------------------------------------------------------------------------------------
  E_PROGRESS.PROGRESS_OCCUPIED:
    CASE _nSubState
    OF
      E_PROGRESS.PROGRESS_INIT:
        _ChannelCtrl.eCmd             := E_NCI_CTRL.RESET;
        _nSubState                    := E_PROGRESS.PROGRESS_BUSY;

      E_PROGRESS.PROGRESS_BUSY:
        IF (_ChannelState.eState = E_NCI_STATE.RESET + E_PROGRESS.PROGRESS_DONE)
        THEN
          _nSubState                  := E_PROGRESS.PROGRESS_INIT;
          _nState                     := E_PROGRESS.PROGRESS_WORKING;

          IF (_MessageLevel > E_MessageType.eMessageWarning)
          THEN
            _stMsg.eType              := E_MessageType.eMessageInfo;
            _stMsg.eSubdevice         := e_Subdevice.JobBase_StartUp;
            _stMsg.iErrorNumber       := _ChannelState.eState;
            _stMsg.sText              := concat('E_NCI_CTRL.RESET: ', TO_STRING(E_PROGRESS.PROGRESS_DONE));
      
            f_MessageSet(_stMsg);
          END_IF
        END_IF
    END_CASE
  //-------------------------------------------------------------------------------------------------------------
  E_PROGRESS.PROGRESS_WORKING:
    CASE _nSubState
    OF
      E_PROGRESS.PROGRESS_INIT:
        _ChannelCtrl.eCmd             := E_NCI_CTRL.CLEAR_GROUP;
        _nSubState                    := E_PROGRESS.PROGRESS_BUSY;

      E_PROGRESS.PROGRESS_BUSY:
        IF (_ChannelState.eState = E_NCI_STATE.CLEAR_GROUP + E_PROGRESS.PROGRESS_DONE)
        THEN
          _nSubState                  := E_PROGRESS.PROGRESS_INIT;
          _nState                     := E_PROGRESS.PROGRESS_STILL_WORKING;

          IF (_MessageLevel > E_MessageType.eMessageWarning)
          THEN
            _stMsg.eType              := E_MessageType.eMessageInfo;
            _stMsg.eSubdevice         := e_Subdevice.NciStartUp;
            _stMsg.iErrorNumber       := _ChannelState.eState;
            _stMsg.sText              := concat('E_NCI_CTRL.CLEAR_GROUP: ', TO_STRING(E_PROGRESS.PROGRESS_DONE));
      
            f_MessageSet(_stMsg);
          END_IF
        END_IF
    END_CASE
  //-------------------------------------------------------------------------------------------------------------
  E_PROGRESS.PROGRESS_STILL_WORKING:
    _nState                           := E_PROGRESS.PROGRESS_DONE;

    IF (_MessageLevel > E_MessageType.eMessageError)
    THEN
      _stMsg.eType                    := E_MessageType.eMessageInfo;
      _stMsg.eSubdevice               := e_Subdevice.NciStartUp;
      _stMsg.iErrorNumber             := 0;
      _stMsg.sText                    := concat(' : ', TO_STRING(_nState));

      f_MessageSet(_stMsg);
    END_IF
END_CASE
//---------------------------------------------------------------------------------------------------------------
Unit_Startup                          := _nState;
//---------------------------------------------------------------------------------------------------------------
END_METHOD

END_FUNCTION_BLOCK

// ---- _MSG/f_MessageSet.TcPOU
FUNCTION f_MessageSet : BOOL
VAR_INPUT
  stMessage     : ST_Message;
END_VAR
VAR
  _uiIndex      : UINT;
  _MainDevice   : e_Device;
  _nModRes      : UDINT;     // residual after modulo
END_VAR

stMessage.tTime                     := GVL_MSG_XTS.sLocalTime;

// why here? so all calls to this function may stay the same
_nModRes                            := stMessage.eDevice MOD e_Device.General;
_MainDevice                         := stMessage.eDevice - _nModRes;

CASE _MainDevice
OF
  //--------------------------------------------------------------------------------
  e_device.DataProduct:
    // this is your data, if you choose to use this message system
    FOR _uiIndex := 1 TO GVL_MSG_XTS.MAX_MESSAGE
    DO
      IF (GVL_MSG_XTS.ProductMessages[_uiIndex].eType = e_MessageType.eMessageEmpty)
      THEN
        GVL_MSG_XTS.ProductMessages[_uiIndex]      := stMessage;
        GVL_MSG_XTS.MessageProductIndex            := _uiIndex;
        EXIT;
      END_IF
    END_FOR
  
    IF (stMessage.eType = E_MessageType.eMessageError)
    THEN
      // in case of error: increment counter
      GVL_MSG_XTS.MessageProductError              := GVL_MSG_XTS.MessageProductError + 1;
    END_IF
  //--------------------------------------------------------------------------------
  e_Device.Process,
  e_Device.Application:
    FOR _uiIndex := 1 TO GVL_MSG_XTS.MAX_MESSAGE
    DO
      IF (GVL_MSG_XTS.ApplicationMessages[_uiIndex].eType = e_MessageType.eMessageEmpty)
      THEN
        GVL_MSG_XTS.ApplicationMessages[_uiIndex]  := stMessage;    // yes, we grab global values directly, only here
        GVL_MSG_XTS.MessageApplicationIndex        := _uiIndex;
        EXIT;
      END_IF
    END_FOR
    IF (stMessage.eType = E_MessageType.eMessageError)
    THEN
      // in case of error: increment counter
      GVL_MSG_XTS.MessageApplicationError          := GVL_MSG_XTS.MessageApplicationError + 1;
    END_IF
  //--------------------------------------------------------------------------------
  e_Device.MetricsXts:
    FOR _uiIndex := 1 TO GVL_MSG_XTS.MAX_MESSAGE
    DO
      IF (GVL_MSG_XTS.MetricsMessages[_uiIndex].eType = e_MessageType.eMessageEmpty)
      THEN
        GVL_MSG_XTS.MetricsMessages[_uiIndex]      := stMessage;    // yes, we grab global values directly, only here
        GVL_MSG_XTS.MessageMetricsIndex            := _uiIndex;
        EXIT;
      END_IF
    END_FOR
    IF (stMessage.eType = E_MessageType.eMessageError)
    THEN
      // in case of error: increment counter
      GVL_MSG_XTS.MessageMetricsError              := GVL_MSG_XTS.MessageMetricsError + 1;
    END_IF
  //--------------------------------------------------------------------------------
  e_Device.MetricsAxis:
    FOR _uiIndex := 1 TO GVL_MSG_XTS.MAX_MESSAGE
    DO
      IF (GVL_MSG_AXIS.MetricMessages[_uiIndex].eType = e_MessageType.eMessageEmpty)
      THEN
        GVL_MSG_AXIS.MetricMessages[_uiIndex]  := stMessage;    // yes, we grab global values directly, only here
        GVL_MSG_AXIS.MessageMetricIndex        := _uiIndex;
        EXIT;
      END_IF
    END_FOR
    IF (stMessage.eType = E_MessageType.eMessageError)
    THEN
      // in case of error: increment counter
      GVL_MSG_AXIS.MessageMetricError          := GVL_MSG_AXIS.MessageMetricError + 1;
    END_IF
  //--------------------------------------------------------------------------------
  e_Device.Axis,
  e_Device.XfcAxis,
  e_device.XfcTouchProbe,
  e_device.XfcTriggerBox,
  e_Device.Camming,
  e_device.NciChannel,
  e_device.NciChannelCtrl:
    FOR _uiIndex := 1 TO GVL_MSG_XTS.MAX_MESSAGE
    DO
      IF (GVL_MSG_AXIS.MotionMessages[_uiIndex].eType = e_MessageType.eMessageEmpty)
      THEN
        GVL_MSG_AXIS.MotionMessages[_uiIndex]  := stMessage;    // yes, we grab global values directly, only here
        GVL_MSG_AXIS.MessageMotionIndex        := _uiIndex;
        EXIT;
      END_IF
    END_FOR
    IF (stMessage.eType = E_MessageType.eMessageError)
    THEN
      // in case of error: increment counter
      GVL_MSG_AXIS.MessageMotionError           := GVL_MSG_AXIS.MessageMotionError + 1;
    END_IF
  //--------------------------------------------------------------------------------
ELSE
  CASE stMessage.eDevice
  OF
    Device_MainApplication,
    Device_XmlData,              
    Device_Utilities:
      FOR _uiIndex := 1 TO GVL_MSG_XTS.MAX_MESSAGE
      DO
        IF (GVL_MSG_XTS.ApplicationMessages[_uiIndex].eType = e_MessageType.eMessageEmpty)
        THEN
          GVL_MSG_XTS.ApplicationMessages[_uiIndex]:= stMessage;    // yes, we grab global values directly, only here
          GVL_MSG_XTS.MessageApplicationIndex      := _uiIndex;
          EXIT;
        END_IF
      END_FOR
      IF (stMessage.eType = E_MessageType.eMessageError)
      THEN
        // in case of error: increment counter
        GVL_MSG_XTS.MessageApplicationError        := GVL_MSG_XTS.MessageApplicationError + 1;
      END_IF

    Device_MainAxis,
    Device_Nci,
    Device_Cam,
    Device_Functions,
    Device_FlyingSaw,
    Device_ParameterSelector:     // PLC_MOTION
      FOR _uiIndex := 1 TO GVL_MSG_XTS.MAX_MESSAGE
      DO
        IF (GVL_MSG_AXIS.MotionMessages[_uiIndex].eType = e_MessageType.eMessageEmpty)
        THEN
          GVL_MSG_AXIS.MotionMessages[_uiIndex]:= stMessage;    // yes, we grab global values directly, only here
          GVL_MSG_AXIS.MessageMotionIndex      := _uiIndex;
          EXIT;
        END_IF
      END_FOR
      IF (stMessage.eType = E_MessageType.eMessageError)
      THEN
        // in case of error: increment counter
        GVL_MSG_AXIS.MessageMotionError        := GVL_MSG_AXIS.MessageMotionError + 1;
      END_IF

    Device_Main,
    Device_MoverSelector:
      FOR _uiIndex := 1 TO GVL_MSG_XTS.MAX_MESSAGE
      DO
        IF (GVL_MSG_XTS.TransportMessages[_uiIndex].eType = e_MessageType.eMessageEmpty)
        THEN
          GVL_MSG_XTS.TransportMessages[_uiIndex]  := stMessage;
          GVL_MSG_XTS.MessageTransportIndex        := _uiIndex;
          EXIT;
        END_IF
      END_FOR
  ELSE    
    //--------------------------------------------------------------------------------
    FOR _uiIndex := 1 TO GVL_MSG_XTS.MAX_MESSAGE
    DO
      IF (GVL_MSG_XTS.TransportMessages[_uiIndex].eType = e_MessageType.eMessageEmpty)
      THEN
        GVL_MSG_XTS.TransportMessages[_uiIndex]    := stMessage;
        GVL_MSG_XTS.MessageTransportIndex          := _uiIndex;
        EXIT;
      END_IF
    END_FOR
  
    IF (stMessage.eType = E_MessageType.eMessageError)
    THEN
      // in case of error: increment counter
      GVL_MSG_XTS.MessageTransportError := GVL_MSG_XTS.MessageTransportError + 1;
    END_IF
  END_CASE
END_CASE

END_FUNCTION

// ---- _MSG/class/fb_MessageDataCtrl.TcPOU
FUNCTION_BLOCK fb_MessageDataCtrl EXTENDS fb_MessageData
VAR
  _stCtrl       : REFERENCE TO ST_MESSAGE_CTRL;
  _stState      : REFERENCE TO ST_MESSAGE_STATE;

  _eCmd,
  _eCmdOld      : E_MESSAGE_CTRL;

  _eResult,
  _eJobResult   : E_PROGRESS;

  _eState       : E_MESSAGE_STATE;

END_VAR

//-----------------------------------------------------------------------------
// check pointers
//-----------------------------------------------------------------------------
IF NOT Check()
THEN
  _eResult                      := E_PROGRESS.PROGRESS_ERROR;
  RETURN;
END_IF
//-----------------------------------------------------------------------------
// check date
// new message file for a new day
//-----------------------------------------------------------------------------
IF (FolderDate(_dtLocalTime) <> _sFolderDate)
THEN
  _bFileCreated                 := FALSE;
END_IF
//-----------------------------------------------------------------------------
//----------------------------------------------------------------------------- 
// copy to local for debug
_eCmd                         := _stCtrl.Cmd;

// cyclic check for command change
// get state for cmd
IF (_eCmd <> _eCmdOld)
THEN
  // get matching sdtate for Ctrl.Cmd
  _eState                     := Cmd(_eCmd);
  _eCmdOld                    := _eCmd;
END_IF


CASE _eResult
OF
  E_PROGRESS.PROGRESS_INVALID:
    _stState.State            := E_MESSAGE_STATE.MSG_STATE_NULL;

  E_PROGRESS.PROGRESS_ERROR:
    _stState.State            := _eState + E_PROGRESS.PROGRESS_ERROR;

  E_PROGRESS.PROGRESS_DONE:
    _stState.State            := _eState + E_PROGRESS.PROGRESS_DONE;

ELSE
  // work in progress
  // update progress for extern use
  _stState.State              := _eState + _eResult;

  CASE _eState
  OF
    E_MESSAGE_STATE.MSG_STATE_INIT:
      _eResult                := BuildFolder(TRUE);


    E_MESSAGE_STATE.MSG_STATE_IDLE:
      IF (_nMsgIndex < GVL_MSG_AXIS.MAX_MESSAGE - GVL_MSG_AXIS.MAX_MESSAGE/10)
      THEN
        _eResult              := E_PROGRESS.PROGRESS_WORKING;
      ELSE
        _eResult              := E_PROGRESS.PROGRESS_DONE;
        _nMsgIndex            := 0;
        // copy from attached list to local
        memcpy(ADR(_aWriteList), _pMsgList, SIZEOF(_aWriteList));
        // clear attached list
        memset(_pMsgList, 0, SIZEOF(_aWriteList));
      END_IF


    E_MESSAGE_STATE.MSG_STATE_WRITE:
      _eResult                := BuildFileData(TRUE);

  ELSE
      _eResult               := E_PROGRESS.PROGRESS_INVALID;
  END_CASE
END_CASE

METHOD BuildFileData : e_progress
VAR_INPUT
  Execute     : BOOL;
END_VAR
VAR_INST
  _nErrorId   : UDINT;
  _eState,
  _eRes       : E_PROGRESS;
  _eFlow      : E_MESSAGE_FLOW;

  _nStringLength  : UINT;
END_VAR
//-----------------------------------------------------------------------------
IF NOT Execute 
THEN
  _eRes                           := WriteData(FALSE);
	_eState                         := E_PROGRESS.PROGRESS_INIT; 
END_IF 
//-----------------------------------------------------------------------------
IF NOT Check() 
THEN 
	BuildFileData                   := E_PROGRESS.PROGRESS_ERROR; 
	RETURN; 
END_IF
//-----------------------------------------------------------------------------
//-----------------------------------------------------------------------------
CASE _eState
OF
  E_PROGRESS.PROGRESS_INIT:
    IF Execute
    THEN
      _nErrorId                   := 0;
      _iStart 	                  := 1;
      _iEnd 		                  := SEL((_nMsgIndex > GVL_MSG_AXIS.MAX_MESSAGE-1),
                                          _nMsgIndex,
                                          GVL_MSG_AXIS.MAX_MESSAGE);

      memset(ADR(_sWriteData),0,SIZEOF(_sWriteData));

      _eState                     := E_PROGRESS.PROGRESS_BUSY;
      _eFlow                      := E_MESSAGE_FLOW.MSG_FLOW_LINE_START;
    END_IF
END_CASE
//-----------------------------------------------------------------------------
//-----------------------------------------------------------------------------
CASE _eState
OF
  E_PROGRESS.PROGRESS_BUSY:
  CASE _eFlow
  OF
    E_MESSAGE_FLOW.MSG_FLOW_LINE_START:
      _nErrIndex                  := 0; // rise and shine, all quarrels erased but not forgotten
      _nMsgIndex                  := 0;
  
      // copy from attached list to local
      memcpy(ADR(_aWriteList), _pMsgList, SIZEOF(_aWriteList));
  
      // clear attached list
      memset(_pMsgList, 0, SIZEOF(_aWriteList));


      _eFlow                      := E_MESSAGE_FLOW.MSG_FLOW_LINE_BUILD;
      _iCount                     := _iStart;
  END_CASE
  CASE _eFlow
  OF
    E_MESSAGE_FLOW.MSG_FLOW_LINE_BUILD:
      _eFlow                      := E_MESSAGE_FLOW.MSG_FLOW_LINE_CHECK;
      IF (_aWriteList[_iCount].eType > E_MessageType.eMessageEmpty)
      THEN
        _sTmp                     := TO_STRING(_aWriteList[_iCount].eType);
        _sTmp                     := Tc2_Standard.CONCAT(_sTmp, _sTab);
        _sTmp                     := Tc2_Standard.CONCAT(_sTmp, _aWriteList[_iCount].tTime);
        _sTmp                     := Tc2_Standard.CONCAT(_sTmp, _sTab);
        _sTmp                     := Tc2_Standard.CONCAT(_sTmp, Device_To_String(_aWriteList[_iCount].eDevice));
        _sTmp                     := Tc2_Standard.CONCAT(_sTmp, _sTab);
        _sTmp                     := Tc2_Standard.CONCAT(_sTmp, TO_STRING(_aWriteList[_iCount].eSubdevice));
        _sTmp                     := Tc2_Standard.CONCAT(_sTmp, _sTab);
        _sTmp                     := Tc2_Standard.CONCAT(_sTmp, TO_STRING(_aWriteList[_iCount].iErrorNumber));
        _sTmp                     := Tc2_Standard.CONCAT(_sTmp, _sTab);
        _sTmp                     := Tc2_Standard.CONCAT(_sTmp, _aWriteList[_iCount].sText);
        _sTmp                     := Tc2_Standard.CONCAT(_sTmp, _sNewLine);
        Builder(ADR(_sTmp), ADR(_sWriteData), StringLen(ADR(_sTmp)));
      END_IF
      _iCount                     := _iCount + 1;
  END_CASE
  CASE _eFlow
  OF
    E_MESSAGE_FLOW.MSG_FLOW_LINE_CHECK:
    IF NOT (_iCount > _iEnd)
    THEN
      _eFlow                      := E_MESSAGE_FLOW.MSG_FLOW_LINE_BUILD;
    ELSE
      _eState                     := E_PROGRESS.PROGRESS_WORKING;
      _eFlow                      := E_MESSAGE_FLOW.MSG_FLOW_WRITE_FILE_BUSY;
    END_IF
  END_CASE
END_CASE
//-----------------------------------------------------------------------------
//-----------------------------------------------------------------------------
CASE _eState
OF
  E_PROGRESS.PROGRESS_WORKING:
  CASE _eFlow
  OF
    E_MESSAGE_FLOW.MSG_FLOW_WRITE_FILE_BUSY:
      _nStringLength              := StringLen(ADR(_sWriteData));
      IF NOT (_nStringLength > 1)
      THEN
        _eState                   := E_PROGRESS.PROGRESS_DONE; 
       _eFlow                     := E_MESSAGE_FLOW.MSG_FLOW_WRITE_FILE_DONE;
      ELSE
        _eFlow                    := E_MESSAGE_FLOW.MSG_FLOW_WRITE_FILE_END;
        _eRes                     := WriteData(FALSE);
      END_IF
  END_CASE
  CASE _eFlow
  OF
    E_MESSAGE_FLOW.MSG_FLOW_WRITE_FILE_END:
      _eRes                       := WriteData(TRUE);

      IF (_eRes = E_PROGRESS.PROGRESS_ERROR)
      THEN
        _eState                   := E_PROGRESS.PROGRESS_ERROR;

      ELSIF (_eRes = E_PROGRESS.PROGRESS_DONE)
      THEN
        _eState                   := E_PROGRESS.PROGRESS_DONE;
        _eFlow                    := E_MESSAGE_FLOW.MSG_FLOW_WRITE_FILE_DONE;
        _eRes                     := WriteData(FALSE);
      END_IF
  END_CASE
END_CASE
//-----------------------------------------------------------------------------
//-----------------------------------------------------------------------------

BuildFileData                     := _eState;
END_METHOD

METHOD BuildFolder : e_progress
VAR_INPUT
  Execute           : BOOL;
END_VAR
VAR_INST
  _nErrorId   : UDINT;
  _eState     : E_PROGRESS;
  _eFlow      : E_MESSAGE_FLOW;
END_VAR
//-----------------------------------------------------------------------------
IF NOT Execute 
THEN 
	_eState                       := E_PROGRESS.PROGRESS_INIT; 
END_IF 
//-----------------------------------------------------------------------------
IF NOT Check() 
THEN 
	BuildFolder                   := E_PROGRESS.PROGRESS_ERROR; 
	RETURN; 
END_IF
//-----------------------------------------------------------------------------
//-----------------------------------------------------------------------------
CASE _eState
OF
  E_PROGRESS.PROGRESS_INIT:
    IF Execute
    THEN
      _nErrorId                 := 0;
      _bFileCreated             := FALSE;

      _sFolderDate              := FolderDate(_dtLocalTime);
      _eState                   := E_PROGRESS.PROGRESS_BUSY;
      _eFlow                    := E_MESSAGE_FLOW.MSG_FLOW_ROOT;
    END_IF
END_CASE
//-----------------------------------------------------------------------------
//-----------------------------------------------------------------------------
CASE _eState
OF
  E_PROGRESS.PROGRESS_BUSY:
  CASE _eFlow
  OF
    E_MESSAGE_FLOW.MSG_FLOW_ROOT:
      _eFlow                    := E_MESSAGE_FLOW.MSG_FLOW_ROOT_CREATE;
      _fbCreateDir.sPathName    := left(_pDirRoot^,len(_pDirRoot^)-1);
      _fbCreateDir(
              bExecute	        := FALSE);
    
    E_MESSAGE_FLOW.MSG_FLOW_ROOT_CREATE:
      (* create root folder *)
      _fbCreateDir(
              bExecute	        := TRUE);
      IF _fbCreateDir.bBusy
      THEN
        _eFlow                  := E_MESSAGE_FLOW.MSG_FLOW_ROOT_CREATE_BUSY;
      END_IF
    
    E_MESSAGE_FLOW.MSG_FLOW_ROOT_CREATE_BUSY:
      _fbCreateDir(
              bExecute	        := TRUE);
      IF NOT _fbCreateDir.bBusy
      THEN
        _eState                 := E_PROGRESS.PROGRESS_PREPARE;
        _eFlow                  := E_MESSAGE_FLOW.MSG_FLOW_FOLDER;
      END_IF
  END_CASE
END_CASE
//-----------------------------------------------------------------------------
//-----------------------------------------------------------------------------
CASE _eState
OF
  E_PROGRESS.PROGRESS_PREPARE:
  CASE _eFlow
  OF
    E_MESSAGE_FLOW.MSG_FLOW_FOLDER:
      _eFlow                    := E_MESSAGE_FLOW.MSG_FLOW_FOLDER_CREATE;
      _sFolderDate              := FolderDate(_dtLocalTime);
      _fbCreateDir.sPathName    := concat(_pDirRoot^, _sFolderDate);
      _fbCreateDir(
              bExecute	        := FALSE);
  
    E_MESSAGE_FLOW.MSG_FLOW_FOLDER_CREATE:
      (* create active folder *)
      _fbCreateDir(
              bExecute	        := TRUE);
      IF _fbCreateDir.bBusy
      THEN
        _eFlow                  := E_MESSAGE_FLOW.MSG_FLOW_FOLDER_CREATE_BUSY;
      END_IF
    
    E_MESSAGE_FLOW.MSG_FLOW_FOLDER_CREATE_BUSY:
      _fbCreateDir(
              bExecute	        := TRUE);
      IF NOT _fbCreateDir.bBusy
      THEN
        _eState                 := E_PROGRESS.PROGRESS_CHECK;
        _eFlow                  := E_MESSAGE_FLOW.MSG_FLOW_FILE_CREATE_DONE;
        _fbCreateDir(
                bExecute	      := FALSE);
      END_IF
  END_CASE
END_CASE
//-----------------------------------------------------------------------------
//-----------------------------------------------------------------------------
CASE _eState
OF
  E_PROGRESS.PROGRESS_CHECK:
  CASE _eFlow
  OF
    E_MESSAGE_FLOW.MSG_FLOW_FILE_CREATE_DONE:
      _eState                   := E_PROGRESS.PROGRESS_DONE;
      _bFileCreated             := TRUE;

      // build complete file path
      _sTmp                     := concat(concat(_pFileRoot^, _sFolderDate),'.txt');
      _sTmp                     := concat('\', _sTmp);
      _sFilename                := concat(_fbCreateDir.sPathName, _sTmp);
  END_CASE
END_CASE

BuildFolder                     := _eState;
END_METHOD

METHOD Check : BOOL
VAR_INPUT
END_VAR

IF NOT __ISVALIDREF(_stCtrl)
THEN
  _eCheck       := E_MESSAGE_CHECK.MSG_CHECK_INVALID_POINTER_CTRL;
  RETURN;
END_IF

IF NOT __ISVALIDREF(_stState)
THEN
  _eCheck       := E_MESSAGE_CHECK.MSG_CHECK_INVALID_POINTER_STATE;
  RETURN;
END_IF
//-----------------------------------------------------------------
//-----------------------------------------------------------------
IF NOT (_dtLocalTime <> 0)
THEN
  _eCheck       := E_MESSAGE_CHECK.MSG_CHECK_INVALID_POINTER_TIME;
  RETURN;
END_IF

IF NOT (_pMsgList <> 0)
THEN
  _eCheck       := E_MESSAGE_CHECK.MSG_CHECK_INVALID_POINTER_LIST;
  RETURN;
END_IF

IF NOT (_pFileRoot <> 0)
THEN
  _eCheck       := E_MESSAGE_CHECK.MSG_CHECK_INVALID_POINTER_ROOT_FILE;
  RETURN;
END_IF

IF NOT (_pDirRoot <> 0)
THEN
  _eCheck       := E_MESSAGE_CHECK.MSG_CHECK_INVALID_POINTER_ROOT_DIR;
  RETURN;
END_IF

IF NOT __ISVALIDREF(_nMsgIndex)
THEN
  _eCheck       := E_MESSAGE_CHECK.MSG_CHECK_INVALID_POINTER_MSG_IDX;
  RETURN;
END_IF

IF NOT __ISVALIDREF(_nErrIndex)
THEN
  _eCheck       := E_MESSAGE_CHECK.MSG_CHECK_INVALID_POINTER_ERR_IDX;
  RETURN;
END_IF


_eCheck         := E_MESSAGE_CHECK.MSG_CHECK_DONE;
Check           := TRUE;
END_METHOD

METHOD Cmd : e_message_state
VAR_INPUT
  Command     : e_message_ctrl;
END_VAR


CASE Command
OF
  E_MESSAGE_CTRL.MSG_CTRL_NULL:
    _eResult                    := E_PROGRESS.PROGRESS_INVALID;
    Cmd                         := E_MESSAGE_STATE.MSG_STATE_NULL;

  E_MESSAGE_CTRL.MSG_CTRL_INIT:
    _eResult                    := BuildFolder(FALSE);
    Cmd                         := E_MESSAGE_STATE.MSG_STATE_INIT;

  E_MESSAGE_CTRL.MSG_CTRL_IDLE:
    _eResult                    := BuildFileData(FALSE);
    Cmd                         := E_MESSAGE_STATE.MSG_STATE_IDLE;

  E_MESSAGE_CTRL.MSG_CTRL_WRITE:
    _eResult                    := BuildFileData(FALSE);
    Cmd                         := E_MESSAGE_STATE.MSG_STATE_WRITE;
    IF (_nMsgIndex = 0)
    THEN
       // go back to sleep
      _eResult                := E_PROGRESS.PROGRESS_DONE;
    END_IF
ELSE
    //_eResult                    := E_PROGRESS.PROGRESS_ERROR;
    Cmd                         := E_MESSAGE_STATE.MSG_STATE_NULL;
END_CASE
END_METHOD

PROPERTY Ctrl : REFERENCE to ST_MESSAGE_CTRL
SET
_stCtrl ref= Ctrl;
END_SET
END_PROPERTY

PROPERTY FileCreated : bool
GET
FileCreated := _bFileCreated;
END_GET
END_PROPERTY

PROPERTY State : REFERENCE TO ST_MESSAGE_STATE
SET
_stState ref= State;
END_SET
END_PROPERTY

END_FUNCTION_BLOCK

// ---- _MSG/class/fb_MessageData.TcPOU
FUNCTION_BLOCK ABSTRACT fb_MessageData IMPLEMENTS I_MessageData
VAR CONSTANT
{attribute 'hide'}
  STR_LEN       : UDINT := 524_288;
END_VAR
VAR
  _eCheck       : E_MESSAGE_CHECK;            // pointer check state

  _pFileRoot    : POINTER TO STRING(255);     // you decide (example in GVL_MSG.LOG_FILE)
  _pDirRoot     : POINTER TO STRING(255);     // see GVL_MSG.LOG_DIR

  _nMsgIndex    : REFERENCE TO UINT;          // Hypnos IS the only one in the village, if there are more you need more villages
  _nErrIndex    : REFERENCE TO UINT;          // Thanatos, Hypnos stern and more serious brother

  _dtLocalTime  : POINTER TO DT;
  _pMsgList     : POINTER TO ARRAY[1..GVL_MSG_AXIS.MAX_MESSAGE] OF ST_Message; // attach your list here

	_rtrigReset   : Tc2_Standard.R_TRIG;
	_aWriteList   : ARRAY[1..GVL_MSG_AXIS.MAX_MESSAGE] OF ST_Message;
	_sWriteData   : STRING(STR_LEN);
	_sNewLine     : STRING := '$N';
	_sTab         : STRING := '$T';
	_iCount, 
	_iStart, 
	_iEnd         : UINT;

	_fbCreateDir  : Tc2_System.FB_CreateDir;
	_sTmp         : STRING(256);
	_sFilename    : STRING(256);
	_sFolderDate  : STRING;
	_bFileCreated : BOOL;

	_fbFileOpen   : Tc2_System.FB_FileOpen;
	_fbFileWrite  : Tc2_System.FB_FileWrite;
	_fbFileClose  : Tc2_System.FB_FileClose;
END_VAR

METHOD Builder : BOOL // string concat for length > 255
VAR_INPUT
  pInString   : POINTER TO STRING;
  pOutString  : POINTER TO STRING(STR_LEN);
  Length      : UINT;
END_VAR
VAR
  Counter     : UDINT;
  pInWork     : POINTER TO BYTE;
  pOutWork    : POINTER TO BYTE;
END_VAR
pOutWork := pOutString;
pInWork := pInString;
Counter := 0;

(*check termination*)
WHILE (pOutWork^ <> 0) AND
      (Counter < STR_LEN+1)
DO
  Counter := Counter + 1;
  pOutWork := pOutWork + 1;
END_WHILE

(* append only if data fits into output *)
IF (Counter + Length < STR_LEN+1)
THEN

  (* append data *)
  FOR Counter := 1 TO Length
  DO
    pOutWork^ := pInWork^;
    pOutWork := pOutWork + 1;
    pInWork := pInWork + 1;
  END_FOR

  (* terminate *)
  pOutWork := pOutWork + 1;
  pOutWork^ := 0;
END_IF
END_METHOD

METHOD Check : BOOL
VAR_INPUT
END_VAR

IF NOT (_dtLocalTime <> 0)
THEN
  _eCheck       := E_MESSAGE_CHECK.MSG_CHECK_INVALID_POINTER_TIME;
  RETURN;
END_IF

IF NOT (_pMsgList <> 0)
THEN
  _eCheck       := E_MESSAGE_CHECK.MSG_CHECK_INVALID_POINTER_LIST;
  RETURN;
END_IF

IF NOT (_pFileRoot <> 0)
THEN
  _eCheck       := E_MESSAGE_CHECK.MSG_CHECK_INVALID_POINTER_ROOT_FILE;
  RETURN;
END_IF

IF NOT (_pDirRoot <> 0)
THEN
  _eCheck       := E_MESSAGE_CHECK.MSG_CHECK_INVALID_POINTER_ROOT_DIR;
  RETURN;
END_IF

IF NOT __ISVALIDREF(_nMsgIndex)
THEN
  _eCheck       := E_MESSAGE_CHECK.MSG_CHECK_INVALID_POINTER_MSG_IDX;
  RETURN;
END_IF

IF NOT __ISVALIDREF(_nErrIndex)
THEN
  _eCheck       := E_MESSAGE_CHECK.MSG_CHECK_INVALID_POINTER_ERR_IDX;
  RETURN;
END_IF


_eCheck         := E_MESSAGE_CHECK.MSG_CHECK_DONE;
Check           := TRUE;
END_METHOD

METHOD Device_to_String : string
VAR_INPUT
  eMsgDevice    : e_Device;
END_VAR
VAR
  sId                 : STRING := '_ID_';
  nId                 : UDINT;
END_VAR
IF (eMsgDevice < e_device.General)
THEN
  // below general case
  nId := TO_UDINT(eMsgDevice);
  sId := concat(sId, TO_STRING(nId));

  Device_to_String := TO_STRING(eMsgDevice);

ELSE
  IF (eMsgDevice >= e_Device.DataProduct)
  THEN
    nId := eMsgDevice MOD e_Device.DataProduct;
    sId := concat(sId, TO_STRING(nId));
 
    Device_to_String := concat(TO_STRING(e_Device.DataProduct), sId);

  ELSIF (eMsgDevice >= e_Device.Application)
  THEN
    nId := eMsgDevice MOD e_Device.Application;
    sId := concat(sId, TO_STRING(nId));
 
    Device_to_String := concat(TO_STRING(e_Device.Application), sId);

  ELSIF (eMsgDevice >= e_Device.TicketListCtrl)
  THEN
    nId := eMsgDevice MOD e_Device.TicketListCtrl;
    sId := concat(sId, TO_STRING(nId));
 
    Device_to_String := concat(TO_STRING(e_Device.TicketListCtrl), sId);

  ELSIF (eMsgDevice >= e_Device.ProcessListCtrl)
  THEN
    nId := eMsgDevice MOD e_Device.ProcessListCtrl;
    sId := concat(sId, TO_STRING(nId));
 
    Device_to_String := concat(TO_STRING(e_Device.ProcessListCtrl), sId);

  ELSIF (eMsgDevice >= e_Device.Process)
  THEN
    nId := eMsgDevice MOD e_Device.Process;
    sId := concat(sId, TO_STRING(nId));
 
    Device_to_String := concat(TO_STRING(e_Device.Process), sId);

  ELSIF (eMsgDevice >= e_Device.FlyingSaw)
  THEN
    nId := eMsgDevice MOD e_Device.FlyingSaw;
    sId := concat(sId, TO_STRING(nId));
 
    Device_to_String := concat(TO_STRING(e_device.FlyingSaw), sId);

  ELSIF (eMsgDevice >= e_Device.MetricsAxis)
  THEN
    nId := eMsgDevice MOD e_Device.MetricsAxis;
    sId := concat(sId, TO_STRING(nId));
 
    Device_to_String := concat(TO_STRING(e_device.MetricsAxis), sId);

  ELSIF (eMsgDevice >= e_Device.MetricsXts)
  THEN
    nId := eMsgDevice MOD e_Device.MetricsXts;
    sId := concat(sId, TO_STRING(nId));
 
    Device_to_String := concat(TO_STRING(e_device.MetricsXts), sId);

  ELSIF (eMsgDevice >= e_device.XfcAxis)
  THEN
    nId := eMsgDevice MOD e_device.XfcAxis;
    sId := concat(sId, TO_STRING(nId));
 
    Device_to_String := concat(TO_STRING(e_device.XfcAxis), sId);

  ELSIF (eMsgDevice >= e_device.Axis)
  THEN
    nId := eMsgDevice MOD e_device.Axis;
    sId := concat(sId, TO_STRING(nId));
 
    Device_to_String := concat(TO_STRING(e_device.Axis), sId);

  ELSIF (eMsgDevice >= e_device.NciChannelCtrl)
  THEN
    nId := eMsgDevice MOD e_device.NciChannelCtrl;
    sId := concat(sId, TO_STRING(nId));
 
    Device_to_String := concat(TO_STRING(e_device.NciChannelCtrl), sId);

  ELSIF (eMsgDevice >= e_device.NciChannel)
  THEN
    nId := eMsgDevice MOD e_device.NciChannel;
    sId := concat(sId, TO_STRING(nId));
 
    Device_to_String := concat(TO_STRING(e_device.NciChannel), sId);

  ELSIF (eMsgDevice >= e_Device.Camming)
  THEN
    nId := eMsgDevice MOD e_Device.Camming;
    sId := concat(sId, TO_STRING(nId));
 
    Device_to_String := concat(TO_STRING(e_device.Camming), sId);

  ELSIF (eMsgDevice >= e_Device.XtsStation)
  THEN
    nId := eMsgDevice MOD e_Device.XtsStation;
    sId := concat(sId, TO_STRING(nId));
 
    Device_to_String := concat(TO_STRING(e_device.XtsStation), sId);

  ELSIF (eMsgDevice >= e_Device.XfcTouchProbe)
  THEN
    nId := eMsgDevice MOD e_Device.XfcTouchProbe;
    sId := concat(sId, TO_STRING(nId));
 
    Device_to_String := concat(TO_STRING(e_device.XfcTouchProbe), sId);

  ELSIF (eMsgDevice >= e_Device.XfcTriggerBox)
  THEN
    nId := eMsgDevice MOD e_Device.XfcTriggerBox;
    sId := concat(sId, TO_STRING(nId));
 
    Device_to_String := concat(TO_STRING(e_device.XfcTriggerBox), sId);

  ELSIF (eMsgDevice >= e_Device.XtsTransportUnit)
  THEN
    nId := eMsgDevice MOD e_Device.XtsTransportUnit;
    sId := concat(sId, TO_STRING(nId));
 
    Device_to_String := concat(TO_STRING(e_device.XtsTransportUnit), sId);

  ELSIF (eMsgDevice >= e_Device.MoverCtrl)
  THEN
    nId := eMsgDevice MOD e_Device.MoverCtrl;
    sId := concat(sId, TO_STRING(nId));
 
    Device_to_String := concat(TO_STRING(e_device.MoverCtrl), sId);

  ELSIF (eMsgDevice >= e_Device.Mover)
  THEN
    nId := eMsgDevice MOD e_Device.Mover;
    sId := concat(sId, TO_STRING(nId));
 
    Device_to_String := concat(TO_STRING(e_device.Mover), sId);

  ELSIF (eMsgDevice >= e_Device.XpuCtrl)
  THEN
    nId := eMsgDevice MOD e_Device.XpuCtrl;
    sId := concat(sId, TO_STRING(nId));
 
    Device_to_String := concat(TO_STRING(e_device.XpuCtrl), sId);

  ELSIF (eMsgDevice >= e_Device.Xpu)
  THEN
    nId := eMsgDevice MOD e_Device.Xpu;
    sId := concat(sId, TO_STRING(nId));
 
    Device_to_String := concat(TO_STRING(e_device.Xpu), sId);

  ELSIF (eMsgDevice >= e_Device.CaGroup)
  THEN
    nId := eMsgDevice MOD e_Device.CaGroup;
    sId := concat(sId, TO_STRING(nId));
 
    Device_to_String := concat(TO_STRING(e_device.CaGroup), sId);

  ELSIF (eMsgDevice >= e_Device.General)
  THEN
    nId := eMsgDevice MOD e_Device.General;
    sId := concat(sId, TO_STRING(nId));
 
    Device_to_String := concat(TO_STRING(e_device.General), sId);

  ELSE
    Device_to_String := TO_STRING(eMsgDevice);
  END_IF
END_IF
END_METHOD

PROPERTY DirRoot : POINTER to string(255)
SET
_pDirRoot := DirRoot;
END_SET
END_PROPERTY

PROPERTY ErrorIndex : reference to uint
SET
_nErrIndex  REF= ErrorIndex;
END_SET
END_PROPERTY

PROPERTY FileRoot : pointer to string(255)
SET
_pFileRoot := FileRoot;
END_SET
END_PROPERTY

METHOD FolderDate : STRING
VAR_INPUT
	LocalTime   : POINTER TO DT;
END_VAR
VAR
	sTmp        : STRING;
END_VAR
IF NOT (LocalTime <> 0)
THEN
	FolderDate := 'NULL';
	RETURN;
END_IF

sTmp := DT_TO_STRING(LocalTime^);

// cut off #dt literal
sTmp := right(sTmp, len(sTmp)-3);

sTmp := replace(sTmp, '_', 1, 5);
sTmp := replace(sTmp, '_', 1, 8);

sTmp := left(sTmp,10);	// year_month_day

FolderDate := sTmp;
END_METHOD

PROPERTY LocalTime : pointer to DT
SET
_dtLocalTime := LocalTime;
END_SET
END_PROPERTY

PROPERTY MessageIndex : reference to uint
SET
_nMsgIndex   REF= MessageIndex;
END_SET
END_PROPERTY

PROPERTY MsgList : pointer to ARRAY[1..GVL_MSG_AXIS.MAX_MESSAGE] OF st_message
SET
_pMsgList := MsgList;
END_SET
END_PROPERTY

METHOD StringLen : UINT // 	string length for len > 255
VAR_INPUT
  pInString		: POINTER TO STRING(STR_LEN);
END_VAR
VAR
	Counter			: UINT;
	pInWork			: POINTER TO BYTE;
END_VAR
pInWork := pInString;
Counter := 0;

WHILE (pInWork^ <> 0) AND
			(Counter < STR_LEN)
DO
	Counter := Counter + 1;
	pInWork := pInWork + 1;
END_WHILE

StringLen := Counter;
END_METHOD

METHOD WriteData  : e_progress
VAR_INPUT
  bExecute        : BOOL;
END_VAR
VAR_INST
  _eState         : e_progress;
  _bError         : BOOL;
  _nErrorId       : UDINT;
END_VAR
IF NOT bExecute
THEN
  _eState                     := E_PROGRESS.PROGRESS_INIT;
END_IF

CASE _eState 
OF

	E_PROGRESS.PROGRESS_INIT:
		_fbFileOpen.bExecute      := FALSE;
		_fbFileWrite.bExecute	    := FALSE;
		_fbFileClose.bExecute	    := FALSE;

		IF bExecute
		THEN
      _nErrorId               := 0;
      _eState                 := E_PROGRESS.PROGRESS_BUSY;
		END_IF

	E_PROGRESS.PROGRESS_BUSY:
		_fbFileOpen.bExecute      := TRUE;

    IF _fbFileOpen.bError
    THEN
		  _fbFileOpen.bExecute    := FALSE;
      _nErrorId               := _fbFileOpen.nErrId;
      _eState                 := E_PROGRESS.PROGRESS_ERROR;

		ELSIF _fbFileOpen.bBusy
		THEN
      _eState                 := E_PROGRESS.PROGRESS_PREPARE;
		END_IF

	E_PROGRESS.PROGRESS_PREPARE:
		IF NOT _fbFileOpen.bBusy
		THEN
		  _fbFileOpen.bExecute    := FALSE;
			_fbFileWrite.bExecute   := TRUE;
      _eState                 := E_PROGRESS.PROGRESS_STARTUP;
		END_IF

	E_PROGRESS.PROGRESS_STARTUP:
    IF _fbFileWrite.bError
    THEN
			_fbFileWrite.bExecute   := FALSE;
      _nErrorId               := _fbFileWrite.nErrId;
      _eState                 := E_PROGRESS.PROGRESS_ERROR;

		ELSIF _fbFileWrite.bBusy
		THEN
      _eState                 := E_PROGRESS.PROGRESS_CHECK;
		END_IF

	E_PROGRESS.PROGRESS_CHECK:
		IF NOT _fbFileWrite.bBusy
		THEN
			_fbFileWrite.bExecute   := FALSE;
			_fbFileClose.bExecute   := TRUE;
      _eState                 := E_PROGRESS.PROGRESS_OCCUPIED;
		END_IF

	E_PROGRESS.PROGRESS_OCCUPIED:
    IF _fbFileClose.bError
    THEN
			_fbFileClose.bExecute   := FALSE;
      _nErrorId               := _fbFileClose.nErrId;
      _eState                 := E_PROGRESS.PROGRESS_ERROR;

		ELSIF _fbFileClose.bBusy
		THEN
      _eState                 := E_PROGRESS.PROGRESS_WORKING;
		END_IF

	E_PROGRESS.PROGRESS_WORKING:
		IF NOT _fbFileClose.bBusy
		THEN
			_fbFileClose.bExecute   := FALSE;
      _eState                 := E_PROGRESS.PROGRESS_DONE;
		END_IF
END_CASE


_fbFileOpen(
	sNetId:= , 
	sPathName:= _sFilename, 
	nMode:= FOPEN_MODEAPPEND OR FOPEN_MODEPLUS, 
	ePath:= PATH_GENERIC, 
	bExecute:= , 
	tTimeout:= T#10S, 
	bBusy=> , 
	bError=> , 
	nErrId=> , 
	hFile=> );

_fbFileWrite(
	sNetId:= , 
	hFile:= _fbFileOpen.hFile, 
	pWriteBuff:= ADR(_sWriteData), 
	cbWriteLen:= StringLen(ADR(_sWriteData)), 
	bExecute:= , 
	tTimeout:= T#10S, 
	bBusy=> , 
	bError=> , 
	nErrId=> , 
	cbWrite=> );

_fbFileClose(
	sNetId:= , 
	hFile:= _fbFileOpen.hFile, 
	bExecute:= , 
	tTimeout:= T#10S, 
	bBusy=> , 
	bError=> , 
	nErrId=> );

WriteData                     := _eState;
END_METHOD

END_FUNCTION_BLOCK

// ---- _MSG/class/fb_LocalTime.TcPOU
//-----------------------------------------------------------------------------------------------
//
//  As time goes by...
//
//  HAUD 2026 07 23
//  - timezone to match UTC device time.
//-----------------------------------------------------------------------------------------------
FUNCTION_BLOCK fb_LocalTime
VAR
  _eState                 : e_progress;   // self startup state, reaches WORKING when done.
  _stSystemtime           : Tc2_Utilities.TIMESTRUCT;

  _stUtcTime              : Tc2_Utilities.T_FILETIME64; // CPU time as 64bit ULINT, meant to be used for measurement
  _sUtcTime               : STRING;
  _dtUtcTime              : DT;

  _stLocalTime            : Tc2_Utilities.T_FILETIME64; // In every wood, in every spring,there is a different green.
  _sLocalTime             : STRING;
  _dtLocalTime            : DT;

  _eTimeZoneId            : Tc2_Utilities.E_TimeZoneID;
  _stTimeZoneInfo         : Tc2_Utilities.ST_TimeZoneInformation;
  _fbGetTimeZoneInfo      : Tc2_Utilities.FB_GetTimeZoneInformation;
  _fbFileTimeToLocalTime  : Tc2_Utilities.FB_FileTime64ToTzSpecificLocalTime;
  _nErrorId               : UDINT;
  _bError                 : BOOL;
END_VAR

//-----------------------------------------------------------------------------------------------
// infosys: https://infosys.beckhoff.com/english.php?content=../content/1033/tcplclib_tc2_system/3622991755.html&id=6591934602709167291
//-----------------------------------------------------------------------------------------------
// This function can be used to read the operating system timestamp. 
// The timestamp is a 64-bit integer value, with an accuracy of 100 ns, 
// which is updated with every call of the PLC. 
// Among other things, it can be used for timing tasks or time measurements. 
// One unit corresponds to 100 ns. 
// The time represents the number of 100 ns intervals since January 1, 1601 (UTC).
//-----------------------------------------------------------------------------------------------
//-----------------------------------------------------------------------------------------------
_stUtcTime                      := F_GetSystemTime(); // UTC time, no delay --> CPU time direct
//-----------------------------------------------------------------------------------------------
//-----------------------------------------------------------------------------------------------
// build UTC time
_sUtcTime                       := SYSTEMTIME_TO_STRING( FILETIME64_TO_SYSTEMTIME( _stUtcTime ));
_dtUtcTime                      := systemtime_to_dt    ( FILETIME64_TO_SYSTEMTIME( _stUtcTime ));
//-----------------------------------------------------------------------------------------------
//-----------------------------------------------------------------------------------------------
// state machine for getting timezone information and add the offset to UTC time
//-----------------------------------------------------------------------------------------------
CASE _eState
OF
  E_PROGRESS.PROGRESS_INVALID:
    _eState                     := E_PROGRESS.PROGRESS_INIT;
    _fbGetTimeZoneInfo(
                      sNetID    := '', 
                      bExecute  := FALSE,
                      bError    => _bError,
                      nErrID    => _nErrorId, 
                      tzID      => _eTimeZoneId, 
                      tzInfo    => _stTimeZoneInfo);
END_CASE
//---------------------------------------------------------------------------------------------
//---------------------------------------------------------------------------------------------
CASE _eState
OF
  E_PROGRESS.PROGRESS_INIT:
    _fbGetTimeZoneInfo(
                      sNetID    := '', 
                      bExecute  := TRUE,
                      bError    => _bError,
                      nErrID    => _nErrorId, 
                      tzID      => _eTimeZoneId, 
                      tzInfo    => _stTimeZoneInfo);

    IF (_fbGetTimeZoneInfo.bBusy)
    THEN
      _eState                   := E_PROGRESS.PROGRESS_PREPARE;
    END_IF
END_CASE
//---------------------------------------------------------------------------------------------
//---------------------------------------------------------------------------------------------
CASE _eState
OF
  E_PROGRESS.PROGRESS_PREPARE:
    _fbGetTimeZoneInfo(
                      sNetID    := '', 
                      bExecute  := TRUE,
                      bError    => _bError,
                      nErrID    => _nErrorId, 
                      tzID      => _eTimeZoneId, 
                      tzInfo    => _stTimeZoneInfo);

    IF NOT (_fbGetTimeZoneInfo.bBusy)
    THEN
      _fbGetTimeZoneInfo(
                      sNetID    := '', 
                      bExecute  := FALSE);

      _eState                   := E_PROGRESS.PROGRESS_WORKING;
    END_IF
END_CASE
//---------------------------------------------------------------------------------------------
//---------------------------------------------------------------------------------------------
CASE _eState
OF
  E_PROGRESS.PROGRESS_WORKING:
    _fbFileTimeToLocalTime(
                      in        := _stUtcTime, 
                      tzInfo    := _stTimeZoneInfo, 
                      out       => _stLocalTime, 
                      eTzID     => _eTimeZoneId);

  // build local time
  _stSystemtime                 := FILETIME64_TO_SYSTEMTIME( _stLocalTime );
  _sLocalTime                   := SYSTEMTIME_TO_STRING    ( _stSystemtime );
  _dtLocalTime                  := systemtime_to_dt        ( _stSystemtime );


  IF (_stSystemtime.wHour   = 0) AND
     (_stSystemtime.wMinute = 0) AND
     (_stSystemtime.wSecond = 0)
  THEN
    //  The passing seasons are but ripples ever repeated in the long long stream.
    _eState                     := E_PROGRESS.PROGRESS_INIT;
  END_IF
END_CASE
//---------------------------------------------------------------------------------------------
//---------------------------------------------------------------------------------------------

METHOD FolderDate : STRING
VAR_INPUT
	LocalTime   : POINTER TO DT;
END_VAR
VAR
	sTmp        : STRING;
END_VAR
IF NOT (LocalTime <> 0)
THEN
	FolderDate := 'NULL';
	RETURN;
END_IF

sTmp := DT_TO_STRING(LocalTime^);

// cut off #dt literal
sTmp := right(sTmp, len(sTmp)-3);

sTmp := replace(sTmp, '_', 1, 5);
sTmp := replace(sTmp, '_', 1, 8);

sTmp := left(sTmp,10);	// year_month_day

FolderDate := sTmp;
END_METHOD

PROPERTY LocalTime : DT
GET
LocalTime := _dtLocalTime;
END_GET
END_PROPERTY

PROPERTY LocalTimeString : string
GET
IF (len(_sLocalTime) >1)
THEN
  LocalTimeString := _sLocalTime;
ELSE
  LocalTimeString := _sUtcTime;
END_IF
END_GET
END_PROPERTY

PROPERTY State : e_progress
GET
State := _eState;
END_GET
END_PROPERTY

PROPERTY UtcTime : DT
GET
UtcTime := _dtUtcTime;
END_GET
END_PROPERTY

PROPERTY UtcTimeString : string
GET
UtcTimeString := _sUtcTime;
END_GET
END_PROPERTY

END_FUNCTION_BLOCK

// ---- MAPPING/MAPPING_out.TcPOU
PROGRAM MAPPING_out
VAR
  bFirstCycle       : BOOL := TRUE;

  AxisCtrl          : U_AXIS_CTRL;
  AxisMoveData      : U_AXIS_MOVE_DATA;
  AxisMotionOptions : U_AXIS_MOTION_OPTIONS;

  AxisGearInData    : U_AXIS_GEAR_IN;
  AxisHoming        : U_AXIS_HOMING;
  AxisParameterWrt  : U_AXIS_NC_PARAMETER_WRT;

  CamCtrl           : U_CAM_CTRL;
  CamData           : U_CAM_DATA;

  TriggerCtrl       : U_TRIGGER_CTRL;

  TouchCtrl         : U_TOUCH_PROBE_CTRL;

  NciControl        : U_NCI_CTRL;
  NciAxisGroup      : U_NCI_AXIS_ID_GROUP;
  NciRparameters    : U_NCI_R_PARAMETER_Q;


  szAxisPara,
  szAxisHoming,
  szAxisGearData,
  szAxisMotionOptions,
  szAxisMoveData,
  szAxisCtrl          : ARRAY[1..2] OF UDINT;

  szCamCtrl           : ARRAY[1..2] OF UDINT;

  szCtrlTouchProbe,
  szCtrlTrigger       :  ARRAY[1..2] OF UDINT;
END_VAR


IF (bFirstCycle)
THEN
  bFirstCycle             := FALSE;

  szAxisCtrl[1]           := SIZEOF(AxisCtrl);
  szAxisCtrl[2]           := SIZEOF(GVL_AXIS.Ctrl);
  
  szAxisMoveData [1]      := SIZEOF(AxisMoveData);
  szAxisMoveData [2]      := SIZEOF(GVL_AXIS.Data);
  
  szAxisMotionOptions [1] := SIZEOF(AxisMotionOptions);
  szAxisMotionOptions [2] := SIZEOF(GVL_AXIS.MotionOptions);
  
  szAxisGearData [1]      := SIZEOF(AxisGearInData);
  szAxisGearData [2]      := SIZEOF(GVL_AXIS.GearInParameter);
  
  szAxisHoming [1]        := SIZEOF(AxisHoming);
  szAxisHoming [2]        := SIZEOF(GVL_AXIS.HomeParameter);
  
  szAxisPara [1]          := SIZEOF(AxisParameterWrt);
  szAxisPara [2]          := SIZEOF(GVL_AXIS.NcParameterWrt);
  
END_IF

  memcpy(ADR(AxisCtrl),                 ADR(GVL_AXIS.Ctrl),             SIZEOF(AxisCTrl));
  memcpy(ADR(AxisMoveData),             ADR(GVL_AXIS.Data),             SIZEOF(AxisMoveData));
  memcpy(ADR(AxisMotionOptions),        ADR(GVL_AXIS.MotionOptions),    SIZEOF(AxisMotionOptions));
  
  memcpy(ADR(AxisGearInData),           ADR(GVL_AXIS.GearInParameter),  SIZEOF(AxisGearInData));
  memcpy(ADR(AxisHoming),               ADR(GVL_AXIS.HomeParameter),    SIZEOF(AxisHoming));
  memcpy(ADR(AxisParameterWrt),         ADR(GVL_AXIS.NcParameterWrt),   SIZEOF(AxisParameterWrt));

  memcpy(ADR(CamCtrl),                  ADR(GVL_CAM.Ctrl),              SIZEOF(CamCtrl));
  memcpy(ADR(CamData),                  ADR(GVL_CAM.Data),              SIZEOF(CamData));

  memcpy(ADR(NciControl),               ADR(GVL_NCI.ChannelCtrl),       SIZEOF(NciControl));
  memcpy(ADR(NciAxisGroup),             ADR(GVL_NCI.AxisConfig),        SIZEOF(NciAxisGroup));
  memcpy(ADR(NciRparameters),           ADR(GVL_NCI.R_ParameterWrite),  SIZEOF(NciRparameters));

END_PROGRAM

// ---- MAPPING/MAPPING_in.TcPOU
PROGRAM MAPPING_in
VAR
  bFirstCycle           : BOOL := TRUE;

  AxisState             : U_AXIS_STATE;
  AxisInfo              : U_AXIS_INFO;
  AxisParameterRd       : U_AXIS_NC_PARAMETER_RD;

  CamState              : U_CAM_STATE;
  CamInfo               : U_CAM_INFO;

  TriggerState          : U_TRIGGER_STATE;

  TouchState            : U_TOUCH_PROBE_STATE;

  NciState              : U_NCI_STATE;
  NciRparameters        : U_NCI_R_PARAMETER_I;


  szAxisPara,
  szAxisInfo,
  szAxisState           : ARRAY[1..2] OF UDINT;

  szCamInfo,
  szCamData,
  szCamState            : ARRAY[1..2] OF UDINT;

  szStateTouchProbe,
  szStateTrigger	      :  ARRAY[1..2] OF UDINT;
END_VAR


IF (bFirstCycle)
THEN
  bFirstCycle         := FALSE;
  
  szAxisState[1]      := SIZEOF(AxisState);
  szAxisState[2]      := SIZEOF(GVL_AXIS.State);
  
  szAxisInfo [1]      := SIZEOF(AxisInfo);
  szAxisInfo [2]      := SIZEOF(GVL_AXIS.Info);
  
  szAxisPara [1]      := SIZEOF(AxisParameterRd);
  szAxisPara [2]      := SIZEOF(GVL_AXIS.NcParameterRd);
END_IF

  memcpy(ADR(GVL_AXIS.State),             ADR(AxisState),              SIZEOF(AxisState));
  memcpy(ADR(GVL_AXIS.Info),              ADR(AxisInfo),               SIZEOF(AxisInfo));
  memcpy(ADR(GVL_AXIS.NcParameterRd),     ADR(AxisParameterRd),        SIZEOF(AxisParameterRd));

  memcpy(ADR(GVL_CAM.State),              ADR(CamState),               SIZEOF(CamState));
  memcpy(ADR(GVL_CAM.Info),               ADR(CamInfo),                SIZEOF(CamInfo));

  memcpy(ADR(GVL_FUNCTIONS.StateTrigger),    ADR(TriggerState),        SIZEOF(TriggerState));
  memcpy(ADR(GVL_FUNCTIONS.StateTouchProbe), ADR(TouchState),          SIZEOF(TouchState));

  memcpy(ADR(GVL_NCI.ChannelState),       ADR(NciState),               SIZEOF(NciState));
  memcpy(ADR(GVL_NCI.R_ParameterRead),    ADR(NciRparameters),         SIZEOF(NciRparameters));

END_PROGRAM

// ---- _XML/Configuration/fb_Configuration.TcPOU
//---------------------------------------------------------------------------------------------------------------
//
//  fb_Configuration
//
//  HAUD 2023.04.14
//  - base xml integration
//
//  HAUD 2026.04.10.
//  - now extending a base class
//
//  - cyclic OnChange wrapper for xml data 
//      - Ctrl/State
//        1. INIT
//        2. READ / WRITE
//
//  - read  ST_STATION_PARAMETER on demand
//  - write ST_STATION_PARAMETER on demand
//
//---------------------------------------------------------------------------------------------------------------
// This SOFTWARE is provided as an Example by THE PROVIDER "as is" and "with all faults." THE PROVIDER makes no 
// representations or warranties of any kind concerning the safety, suitability, lack of viruses, inaccuracies, 
// typographical errors, or other harmful components of this SOFTWARE. There are inherent dangers in the use of 
// any software, and you are solely responsible for determining whether this SOFTWARE is compatible with your 
// equipment and other software installed on your equipment. You are also solely responsible for the protection 
// of your equipment and backup of your data, and THE PROVIDER will not be liable for any damages you may suffer 
// in connection with using, modifying, or distributing this SOFTWARE.
//---------------------------------------------------------------------------------------------------------------
FUNCTION_BLOCK fb_Configuration EXTENDS fb_XmlBase
VAR
  _stCtrl               : REFERENCE TO ST_DATA_CTRL;
  _stState              : REFERENCE TO ST_DATA_STATE;

  _stConfiguration      : ST_Configuration;
  _pParameter           : POINTER TO ST_CONFIG_PORTAL;
END_VAR
VAR CONSTANT
  FILE_ROOT             : STRING := 'CONFIG_APPLICATION_';
  X_PATH                : STRING := '/config';
END_VAR

//---------------------------------------------------------------------------------------------------------------
//  check pointers from the outside
//---------------------------------------------------------------------------------------------------------------
IF NOT Check() THEN RETURN; END_IF
//---------------------------------------------------------------------------------------------------------------
// always build the internal data pointer
//  - as always: better safe than sorry
//  - leave this bit here, it doesn't cost much and safely addresses the data
//---------------------------------------------------------------------------------------------------------------
_pData                        := ADR    (_stConfiguration);
_nData                        := SIZEOF (_stConfiguration);
_sXpath                       := X_PATH;

// copy to local for debug
_eCmd                         := _stCtrl.Cmd;

// cyclic check for command change
// get state for cmd
IF (_eCmd <> _eCmdOld)
THEN
  // get matching sdtate for Ctrl.Cmd
  _eState                     := Cmd(_eCmd);
  _eCmdOld                    := _eCmd;
END_IF


CASE _eResult
OF
  E_PROGRESS.PROGRESS_INVALID:
    _stState.State            := E_DATA_STATE.NULL;

  E_PROGRESS.PROGRESS_ERROR:
    _stState.State            := _eState + E_PROGRESS.PROGRESS_ERROR;

  E_PROGRESS.PROGRESS_DONE:
    _stState.State            := _eState + E_PROGRESS.PROGRESS_DONE;

ELSE
  // work in progress
  // update progress for extern use
  _stState.State              := _eState + _eResult;

  CASE _eState
  OF
    E_DATA_STATE.INIT:
      _eResult   := _eInit    := CreateFolder(TRUE);

